LIN {X 26.609, Y 67.769, Z 160.75, A 0, B 90, C 0, E1 0, E2 0, E3 0, E4 0} C_DIS
LIN {X 29.432, Y 66.695, Z 160.75, A 0, B 90, C 0, E1 0, E2 0, E3 0, E4 0} C_DIS
LIN {X 32.336, Y 65.861, Z 160.75, A 0, B 90, C 0, E1 0, E2 0, E3 0, E4 0} C_DIS
LIN {X 35.293, Y 65.239, Z 160.75, A 0, B 90, C 0, E1 0, E2 0, E3 0, E4 0} C_DIS
LIN {X 38.28, Y 64.777, Z 160.75, A 0, B 90, C 0, E1 0, E2 0, E3 0, E4 0} C_DIS
LIN {X 41.281, Y 64.423, Z 160.75, A 0, B 90, C 0, E1 0, E2 0, E3 0, E4 0} C_DIS
LIN {X 44.288, Y 64.127, Z 160.75, A 0, B 90, C 0, E1 0, E2 0, E3 0, E4 0} C_DIS
LIN {X 47.298, Y 63.846, Z 160.75, A 0, B 90, C 0, E1 0, E2 0, E3 0, E4 0} C_DIS
LIN {X 50.305, Y 63.548, Z 160.75, A 0, B 90, C 0, E1 0, E2 0, E3 0, E4 0} C_DIS
LIN {X 53.308, Y 63.205, Z 160.75, A 0, B 90, C 0, E1 0, E2 0, E3 0, E4 0} C_DIS
LIN {X 56.302, Y 62.795, Z 160.75, A 0, B 90, C 0, E1 0, E2 0, E3 0, E4 0} C_DIS
LIN {X 59.283, Y 62.3, Z 160.75, A 0, B 90, C 0, E1 0, E2 0, E3 0, E4 0} C_DIS
LIN {X 62.245, Y 61.704, Z 160.75, A 0, B 90, C 0, E1 0, E2 0, E3 0, E4 0} C_DIS
LIN {X 65.182, Y 60.99, Z 160.75, A 0, B 90, C 0, E1 0, E2 0, E3 0, E4 0} C_DIS
LIN {X 68.084, Y 60.146, Z 160.75, A 0, B 90, C 0, E1 0, E2 0, E3 0, E4 0} C_DIS
LIN {X 70.939, Y 59.158, Z 160.75, A 0, B 90, C 0, E1 0, E2 0, E3 0, E4 0} C_DIS
LIN {X 73.737, Y 58.015, Z 160.75, A 0, B 90, C 0, E1 0, E2 0, E3 0, E4 0} C_DIS
LIN {X 76.46, Y 56.707, Z 160.75, A 0, B 90, C 0, E1 0, E2 0, E3 0, E4 0} C_DIS
LIN {X 79.094, Y 55.225, Z 160.75, A 0, B 90, C 0, E1 0, E2 0, E3 0, E4 0} C_DIS
LIN {X 81.618, Y 53.564, Z 160.75, A 0, B 90, C 0, E1 0, E2 0, E3 0, E4 0} C_DIS
LIN {X 84.013, Y 51.722, Z 160.75, A 0, B 90, C 0, E1 0, E2 0, E3 0, E4 0} C_DIS
LIN {X 86.258, Y 49.701, Z 160.75, A 0, B 90, C 0, E1 0, E2 0, E3 0, E4 0} C_DIS
LIN {X 88.328, Y 47.5, Z 160.75, A 0, B 90, C 0, E1 0, E2 0, E3 0, E4 0} C_DIS
LIN {X 90.195, Y 45.125, Z 160.75, A 0, B 90, C 0, E1 0, E2 0, E3 0, E4 0} C_DIS
LIN {X 91.836, Y 42.588, Z 160.75, A 0, B 90, C 0, E1 0, E2 0, E3 0, E4 0} C_DIS
LIN {X 93.229, Y 39.908, Z 160.75, A 0, B 90, C 0, E1 0, E2 0, E3 0, E4 0} C_DIS
LIN {X 94.359, Y 37.106, Z 160.75, A 0, B 90, C 0, E1 0, E2 0, E3 0, E4 0} C_DIS
LIN {X 95.213, Y 34.208, Z 160.75, A 0, B 90, C 0, E1 0, E2 0, E3 0, E4 0} C_DIS
LIN {X 95.79, Y 31.243, Z 160.75, A 0, B 90, C 0, E1 0, E2 0, E3 0, E4 0} C_DIS
LIN {X 96.091, Y 28.237, Z 160.75, A 0, B 90, C 0, E1 0, E2 0, E3 0, E4 0} C_DIS
LIN {X 96.125, Y 25.216, Z 160.75, A 0, B 90, C 0, E1 0, E2 0, E3 0, E4 0} C_DIS
LIN {X 95.904, Y 22.202, Z 160.75, A 0, B 90, C 0, E1 0, E2 0, E3 0, E4 0} C_DIS
LIN {X 95.444, Y 19.216, Z 160.75, A 0, B 90, C 0, E1 0, E2 0, E3 0, E4 0} C_DIS
LIN {X 94.762, Y 16.273, Z 160.75, A 0, B 90, C 0, E1 0, E2 0, E3 0, E4 0} C_DIS
LIN {X 93.877, Y 13.384, Z 160.75, A 0, B 90, C 0, E1 0, E2 0, E3 0, E4 0} C_DIS
LIN {X 92.806, Y 10.558, Z 160.75, A 0, B 90, C 0, E1 0, E2 0, E3 0, E4 0} C_DIS
LIN {X 91.571, Y 7.8, Z 160.75, A 0, B 90, C 0, E1 0, E2 0, E3 0, E4 0} C_DIS
LIN {X 90.195, Y 5.11, Z 160.75, A 0, B 90, C 0, E1 0, E2 0, E3 0, E4 0} C_DIS
LIN {X 88.691, Y 2.489, Z 160.75, A 0, B 90, C 0, E1 0, E2 0, E3 0, E4 0} C_DIS
LIN {X 87.109, Y 0, Z 160.75, A 0, B 90, C 0, E1 0, E2 0, E3 0, E4 0} C_DIS
LIN {X 85.255, Y -2.058, Z 160.75, A 0, B 90, C 0, E1 0, E2 0, E3 0, E4 0} C_DIS
LIN {X 83.459, Y -4.487, Z 160.75, A 0, B 90, C 0, E1 0, E2 0, E3 0, E4 0} C_DIS
LIN {X 81.625, Y -6.889, Z 160.75, A 0, B 90, C 0, E1 0, E2 0, E3 0, E4 0} C_DIS
LIN {X 79.745, Y -9.255, Z 160.75, A 0, B 90, C 0, E1 0, E2 0, E3 0, E4 0} C_DIS
LIN {X 77.844, Y -11.605, Z 160.75, A 0, B 90, C 0, E1 0, E2 0, E3 0, E4 0} C_DIS
LIN {X 75.949, Y -13.959, Z 160.75, A 0, B 90, C 0, E1 0, E2 0, E3 0, E4 0} C_DIS
LIN {X 74.087, Y -16.339, Z 160.75, A 0, B 90, C 0, E1 0, E2 0, E3 0, E4 0} C_DIS
LIN {X 72.293, Y -18.771, Z 160.75, A 0, B 90, C 0, E1 0, E2 0, E3 0, E4 0} C_DIS
LIN {X 70.608, Y -21.279, Z 160.75, A 0, B 90, C 0, E1 0, E2 0, E3 0, E4 0} C_DIS
LIN {X 69.084, Y -23.889, Z 160.75, A 0, B 90, C 0, E1 0, E2 0, E3 0, E4 0} C_DIS
LIN {X 67.769, Y -26.609, Z 160.75, A 0, B 90, C 0, E1 0, E2 0, E3 0, E4 0} C_DIS
LIN {X 66.695, Y -29.432, Z 160.75, A 0, B 90, C 0, E1 0, E2 0, E3 0, E4 0} C_DIS
LIN {X 65.861, Y -32.336, Z 160.75, A 0, B 90, C 0, E1 0, E2 0, E3 0, E4 0} C_DIS
LIN {X 65.239, Y -35.293, Z 160.75, A 0, B 90, C 0, E1 0, E2 0, E3 0, E4 0} C_DIS
LIN {X 64.777, Y -38.28, Z 160.75, A 0, B 90, C 0, E1 0, E2 0, E3 0, E4 0} C_DIS
LIN {X 64.423, Y -41.281, Z 160.75, A 0, B 90, C 0, E1 0, E2 0, E3 0, E4 0} C_DIS
LIN {X 64.127, Y -44.288, Z 160.75, A 0, B 90, C 0, E1 0, E2 0, E3 0, E4 0} C_DIS
LIN {X 63.846, Y -47.298, Z 160.75, A 0, B 90, C 0, E1 0, E2 0, E3 0, E4 0} C_DIS
LIN {X 63.548, Y -50.305, Z 160.75, A 0, B 90, C 0, E1 0, E2 0, E3 0, E4 0} C_DIS
LIN {X 63.205, Y -53.308, Z 160.75, A 0, B 90, C 0, E1 0, E2 0, E3 0, E4 0} C_DIS
LIN {X 62.795, Y -56.302, Z 160.75, A 0, B 90, C 0, E1 0, E2 0, E3 0, E4 0} C_DIS
LIN {X 62.3, Y -59.283, Z 160.75, A 0, B 90, C 0, E1 0, E2 0, E3 0, E4 0} C_DIS
LIN {X 61.704, Y -62.245, Z 160.75, A 0, B 90, C 0, E1 0, E2 0, E3 0, E4 0} C_DIS
LIN {X 60.99, Y -65.182, Z 160.75, A 0, B 90, C 0, E1 0, E2 0, E3 0, E4 0} C_DIS
LIN {X 60.146, Y -68.084, Z 160.75, A 0, B 90, C 0, E1 0, E2 0, E3 0, E4 0} C_DIS
LIN {X 59.158, Y -70.939, Z 160.75, A 0, B 90, C 0, E1 0, E2 0, E3 0, E4 0} C_DIS
LIN {X 58.015, Y -73.737, Z 160.75, A 0, B 90, C 0, E1 0, E2 0, E3 0, E4 0} C_DIS
LIN {X 56.707, Y -76.46, Z 160.75, A 0, B 90, C 0, E1 0, E2 0, E3 0, E4 0} C_DIS
LIN {X 55.225, Y -79.094, Z 160.75, A 0, B 90, C 0, E1 0, E2 0, E3 0, E4 0} C_DIS
LIN {X 53.564, Y -81.618, Z 160.75, A 0, B 90, C 0, E1 0, E2 0, E3 0, E4 0} C_DIS
LIN {X 51.722, Y -84.013, Z 160.75, A 0, B 90, C 0, E1 0, E2 0, E3 0, E4 0} C_DIS
LIN {X 49.701, Y -86.258, Z 160.75, A 0, B 90, C 0, E1 0, E2 0, E3 0, E4 0} C_DIS
LIN {X 47.5, Y -88.328, Z 160.75, A 0, B 90, C 0, E1 0, E2 0, E3 0, E4 0} C_DIS
LIN {X 45.125, Y -90.195, Z 160.75, A 0, B 90, C 0, E1 0, E2 0, E3 0, E4 0} C_DIS
LIN {X 42.588, Y -91.836, Z 160.75, A 0, B 90, C 0, E1 0, E2 0, E3 0, E4 0} C_DIS
LIN {X 39.908, Y -93.229, Z 160.75, A 0, B 90, C 0, E1 0, E2 0, E3 0, E4 0} C_DIS
LIN {X 37.106, Y -94.359, Z 160.75, A 0, B 90, C 0, E1 0, E2 0, E3 0, E4 0} C_DIS
LIN {X 34.208, Y -95.213, Z 160.75, A 0, B 90, C 0, E1 0, E2 0, E3 0, E4 0} C_DIS
LIN {X 31.243, Y -95.79, Z 160.75, A 0, B 90, C 0, E1 0, E2 0, E3 0, E4 0} C_DIS
LIN {X 28.237, Y -96.091, Z 160.75, A 0, B 90, C 0, E1 0, E2 0, E3 0, E4 0} C_DIS
LIN {X 25.216, Y -96.125, Z 160.75, A 0, B 90, C 0, E1 0, E2 0, E3 0, E4 0} C_DIS
LIN {X 22.202, Y -95.904, Z 160.75, A 0, B 90, C 0, E1 0, E2 0, E3 0, E4 0} C_DIS
LIN {X 19.216, Y -95.444, Z 160.75, A 0, B 90, C 0, E1 0, E2 0, E3 0, E4 0} C_DIS
LIN {X 16.273, Y -94.762, Z 160.75, A 0, B 90, C 0, E1 0, E2 0, E3 0, E4 0} C_DIS
LIN {X 13.384, Y -93.877, Z 160.75, A 0, B 90, C 0, E1 0, E2 0, E3 0, E4 0} C_DIS
LIN {X 10.558, Y -92.806, Z 160.75, A 0, B 90, C 0, E1 0, E2 0, E3 0, E4 0} C_DIS
LIN {X 7.8, Y -91.571, Z 160.75, A 0, B 90, C 0, E1 0, E2 0, E3 0, E4 0} C_DIS
LIN {X 5.11, Y -90.195, Z 160.75, A 0, B 90, C 0, E1 0, E2 0, E3 0, E4 0} C_DIS
LIN {X 2.489, Y -88.691, Z 160.75, A 0, B 90, C 0, E1 0, E2 0, E3 0, E4 0} C_DIS
LIN {X 0, Y -87.109, Z 160.75, A 0, B 90, C 0, E1 0, E2 0, E3 0, E4 0} C_DIS
LIN {X -2.058, Y -85.255, Z 160.75, A 0, B 90, C 0, E1 0, E2 0, E3 0, E4 0} C_DIS
LIN {X -4.487, Y -83.459, Z 160.75, A 0, B 90, C 0, E1 0, E2 0, E3 0, E4 0} C_DIS
LIN {X -6.889, Y -81.625, Z 160.75, A 0, B 90, C 0, E1 0, E2 0, E3 0, E4 0} C_DIS
LIN {X -9.255, Y -79.745, Z 160.75, A 0, B 90, C 0, E1 0, E2 0, E3 0, E4 0} C_DIS
LIN {X -11.605, Y -77.844, Z 160.75, A 0, B 90, C 0, E1 0, E2 0, E3 0, E4 0} C_DIS
LIN {X -13.959, Y -75.949, Z 160.75, A 0, B 90, C 0, E1 0, E2 0, E3 0, E4 0} C_DIS
LIN {X -16.339, Y -74.087, Z 160.75, A 0, B 90, C 0, E1 0, E2 0, E3 0, E4 0} C_DIS
LIN {X -18.771, Y -72.293, Z 160.75, A 0, B 90, C 0, E1 0, E2 0, E3 0, E4 0} C_DIS
LIN {X -21.279, Y -70.608, Z 160.75, A 0, B 90, C 0, E1 0, E2 0, E3 0, E4 0} C_DIS
LIN {X -23.889, Y -69.084, Z 160.75, A 0, B 90, C 0, E1 0, E2 0, E3 0, E4 0} C_DIS
LIN {X -26.609, Y -67.769, Z 160.75, A 0, B 90, C 0, E1 0, E2 0, E3 0, E4 0} C_DIS
LIN {X -29.432, Y -66.695, Z 160.75, A 0, B 90, C 0, E1 0, E2 0, E3 0, E4 0} C_DIS
LIN {X -32.336, Y -65.861, Z 160.75, A 0, B 90, C 0, E1 0, E2 0, E3 0, E4 0} C_DIS
LIN {X -35.293, Y -65.239, Z 160.75, A 0, B 90, C 0, E1 0, E2 0, E3 0, E4 0} C_DIS
LIN {X -38.28, Y -64.777, Z 160.75, A 0, B 90, C 0, E1 0, E2 0, E3 0, E4 0} C_DIS
LIN {X -41.281, Y -64.423, Z 160.75, A 0, B 90, C 0, E1 0, E2 0, E3 0, E4 0} C_DIS
LIN {X -44.288, Y -64.127, Z 160.75, A 0, B 90, C 0, E1 0, E2 0, E3 0, E4 0} C_DIS
LIN {X -47.298, Y -63.846, Z 160.75, A 0, B 90, C 0, E1 0, E2 0, E3 0, E4 0} C_DIS
LIN {X -50.305, Y -63.548, Z 160.75, A 0, B 90, C 0, E1 0, E2 0, E3 0, E4 0} C_DIS
LIN {X -53.308, Y -63.205, Z 160.75, A 0, B 90, C 0, E1 0, E2 0, E3 0, E4 0} C_DIS
LIN {X -56.302, Y -62.795, Z 160.75, A 0, B 90, C 0, E1 0, E2 0, E3 0, E4 0} C_DIS
LIN {X -59.283, Y -62.3, Z 160.75, A 0, B 90, C 0, E1 0, E2 0, E3 0, E4 0} C_DIS
LIN {X -62.245, Y -61.704, Z 160.75, A 0, B 90, C 0, E1 0, E2 0, E3 0, E4 0} C_DIS
LIN {X -65.182, Y -60.99, Z 160.75, A 0, B 90, C 0, E1 0, E2 0, E3 0, E4 0} C_DIS
LIN {X -68.084, Y -60.146, Z 160.75, A 0, B 90, C 0, E1 0, E2 0, E3 0, E4 0} C_DIS
LIN {X -70.939, Y -59.158, Z 160.75, A 0, B 90, C 0, E1 0, E2 0, E3 0, E4 0} C_DIS
LIN {X -73.737, Y -58.015, Z 160.75, A 0, B 90, C 0, E1 0, E2 0, E3 0, E4 0} C_DIS
LIN {X -76.46, Y -56.707, Z 160.75, A 0, B 90, C 0, E1 0, E2 0, E3 0, E4 0} C_DIS
LIN {X -79.094, Y -55.225, Z 160.75, A 0, B 90, C 0, E1 0, E2 0, E3 0, E4 0} C_DIS
LIN {X -81.618, Y -53.564, Z 160.75, A 0, B 90, C 0, E1 0, E2 0, E3 0, E4 0} C_DIS
LIN {X -84.013, Y -51.722, Z 160.75, A 0, B 90, C 0, E1 0, E2 0, E3 0, E4 0} C_DIS
LIN {X -86.258, Y -49.701, Z 160.75, A 0, B 90, C 0, E1 0, E2 0, E3 0, E4 0} C_DIS
LIN {X -88.328, Y -47.5, Z 160.75, A 0, B 90, C 0, E1 0, E2 0, E3 0, E4 0} C_DIS
LIN {X -90.195, Y -45.125, Z 160.75, A 0, B 90, C 0, E1 0, E2 0, E3 0, E4 0} C_DIS
LIN {X -91.836, Y -42.588, Z 160.75, A 0, B 90, C 0, E1 0, E2 0, E3 0, E4 0} C_DIS
LIN {X -93.229, Y -39.908, Z 160.75, A 0, B 90, C 0, E1 0, E2 0, E3 0, E4 0} C_DIS
LIN {X -94.359, Y -37.106, Z 160.75, A 0, B 90, C 0, E1 0, E2 0, E3 0, E4 0} C_DIS
LIN {X -95.213, Y -34.208, Z 160.75, A 0, B 90, C 0, E1 0, E2 0, E3 0, E4 0} C_DIS
LIN {X -95.79, Y -31.243, Z 160.75, A 0, B 90, C 0, E1 0, E2 0, E3 0, E4 0} C_DIS
LIN {X -96.091, Y -28.237, Z 160.75, A 0, B 90, C 0, E1 0, E2 0, E3 0, E4 0} C_DIS
LIN {X -96.125, Y -25.216, Z 160.75, A 0, B 90, C 0, E1 0, E2 0, E3 0, E4 0} C_DIS
LIN {X -95.904, Y -22.202, Z 160.75, A 0, B 90, C 0, E1 0, E2 0, E3 0, E4 0} C_DIS
LIN {X -95.444, Y -19.216, Z 160.75, A 0, B 90, C 0, E1 0, E2 0, E3 0, E4 0} C_DIS
LIN {X -94.762, Y -16.273, Z 160.75, A 0, B 90, C 0, E1 0, E2 0, E3 0, E4 0} C_DIS
LIN {X -93.877, Y -13.384, Z 160.75, A 0, B 90, C 0, E1 0, E2 0, E3 0, E4 0} C_DIS
LIN {X -92.806, Y -10.558, Z 160.75, A 0, B 90, C 0, E1 0, E2 0, E3 0, E4 0} C_DIS
LIN {X -91.571, Y -7.8, Z 160.75, A 0, B 90, C 0, E1 0, E2 0, E3 0, E4 0} C_DIS
LIN {X -90.195, Y -5.11, Z 160.75, A 0, B 90, C 0, E1 0, E2 0, E3 0, E4 0} C_DIS
LIN {X -88.691, Y -2.489, Z 160.75, A 0, B 90, C 0, E1 0, E2 0, E3 0, E4 0} C_DIS
LIN {X -87.509, Y 0, Z 163.25, A 0, B 90, C 0, E1 0, E2 0, E3 0, E4 0} C_DIS
LIN {X -85.636, Y 2.054, Z 163.25, A 0, B 90, C 0, E1 0, E2 0, E3 0, E4 0} C_DIS
LIN {X -83.819, Y 4.483, Z 163.25, A 0, B 90, C 0, E1 0, E2 0, E3 0, E4 0} C_DIS
LIN {X -81.966, Y 6.885, Z 163.25, A 0, B 90, C 0, E1 0, E2 0, E3 0, E4 0} C_DIS
LIN {X -80.069, Y 9.253, Z 163.25, A 0, B 90, C 0, E1 0, E2 0, E3 0, E4 0} C_DIS
LIN {X -78.156, Y 11.608, Z 163.25, A 0, B 90, C 0, E1 0, E2 0, E3 0, E4 0} C_DIS
LIN {X -76.258, Y 13.975, Z 163.25, A 0, B 90, C 0, E1 0, E2 0, E3 0, E4 0} C_DIS
LIN {X -74.403, Y 16.376, Z 163.25, A 0, B 90, C 0, E1 0, E2 0, E3 0, E4 0} C_DIS
LIN {X -72.622, Y 18.832, Z 163.25, A 0, B 90, C 0, E1 0, E2 0, E3 0, E4 0} C_DIS
LIN {X -70.954, Y 21.366, Z 163.25, A 0, B 90, C 0, E1 0, E2 0, E3 0, E4 0} C_DIS
LIN {X -69.45, Y 24.001, Z 163.25, A 0, B 90, C 0, E1 0, E2 0, E3 0, E4 0} C_DIS
LIN {X -68.156, Y 26.744, Z 163.25, A 0, B 90, C 0, E1 0, E2 0, E3 0, E4 0} C_DIS
LIN {X -67.106, Y 29.59, Z 163.25, A 0, B 90, C 0, E1 0, E2 0, E3 0, E4 0} C_DIS
LIN {X -66.295, Y 32.513, Z 163.25, A 0, B 90, C 0, E1 0, E2 0, E3 0, E4 0} C_DIS
LIN {X -65.695, Y 35.486, Z 163.25, A 0, B 90, C 0, E1 0, E2 0, E3 0, E4 0} C_DIS
LIN {X -65.252, Y 38.488, Z 163.25, A 0, B 90, C 0, E1 0, E2 0, E3 0, E4 0} C_DIS
LIN {X -64.912, Y 41.503, Z 163.25, A 0, B 90, C 0, E1 0, E2 0, E3 0, E4 0} C_DIS
LIN {X -64.622, Y 44.523, Z 163.25, A 0, B 90, C 0, E1 0, E2 0, E3 0, E4 0} C_DIS
LIN {X -64.34, Y 47.544, Z 163.25, A 0, B 90, C 0, E1 0, E2 0, E3 0, E4 0} C_DIS
LIN {X -64.029, Y 50.562, Z 163.25, A 0, B 90, C 0, E1 0, E2 0, E3 0, E4 0} C_DIS
LIN {X -63.665, Y 53.574, Z 163.25, A 0, B 90, C 0, E1 0, E2 0, E3 0, E4 0} C_DIS
LIN {X -63.229, Y 56.577, Z 163.25, A 0, B 90, C 0, E1 0, E2 0, E3 0, E4 0} C_DIS
LIN {X -62.704, Y 59.565, Z 163.25, A 0, B 90, C 0, E1 0, E2 0, E3 0, E4 0} C_DIS
LIN {X -62.074, Y 62.533, Z 163.25, A 0, B 90, C 0, E1 0, E2 0, E3 0, E4 0} C_DIS
LIN {X -61.326, Y 65.473, Z 163.25, A 0, B 90, C 0, E1 0, E2 0, E3 0, E4 0} C_DIS
LIN {X -60.446, Y 68.376, Z 163.25, A 0, B 90, C 0, E1 0, E2 0, E3 0, E4 0} C_DIS
LIN {X -59.421, Y 71.232, Z 163.25, A 0, B 90, C 0, E1 0, E2 0, E3 0, E4 0} C_DIS
LIN {X -58.24, Y 74.026, Z 163.25, A 0, B 90, C 0, E1 0, E2 0, E3 0, E4 0} C_DIS
LIN {X -56.893, Y 76.744, Z 163.25, A 0, B 90, C 0, E1 0, E2 0, E3 0, E4 0} C_DIS
LIN {X -55.374, Y 79.37, Z 163.25, A 0, B 90, C 0, E1 0, E2 0, E3 0, E4 0} C_DIS
LIN {X -53.681, Y 81.887, Z 163.25, A 0, B 90, C 0, E1 0, E2 0, E3 0, E4 0} C_DIS
LIN {X -51.817, Y 84.28, Z 163.25, A 0, B 90, C 0, E1 0, E2 0, E3 0, E4 0} C_DIS
LIN {X -49.786, Y 86.534, Z 163.25, A 0, B 90, C 0, E1 0, E2 0, E3 0, E4 0} C_DIS
LIN {X -47.585, Y 88.62, Z 163.25, A 0, B 90, C 0, E1 0, E2 0, E3 0, E4 0} C_DIS
LIN {X -45.213, Y 90.511, Z 163.25, A 0, B 90, C 0, E1 0, E2 0, E3 0, E4 0} C_DIS
LIN {X -42.679, Y 92.178, Z 163.25, A 0, B 90, C 0, E1 0, E2 0, E3 0, E4 0} C_DIS
LIN {X -40, Y 93.599, Z 163.25, A 0, B 90, C 0, E1 0, E2 0, E3 0, E4 0} C_DIS
LIN {X -37.197, Y 94.757, Z 163.25, A 0, B 90, C 0, E1 0, E2 0, E3 0, E4 0} C_DIS
LIN {X -34.295, Y 95.639, Z 163.25, A 0, B 90, C 0, E1 0, E2 0, E3 0, E4 0} C_DIS
LIN {X -31.322, Y 96.242, Z 163.25, A 0, B 90, C 0, E1 0, E2 0, E3 0, E4 0} C_DIS
LIN {X -28.307, Y 96.566, Z 163.25, A 0, B 90, C 0, E1 0, E2 0, E3 0, E4 0} C_DIS
LIN {X -25.274, Y 96.62, Z 163.25, A 0, B 90, C 0, E1 0, E2 0, E3 0, E4 0} C_DIS
LIN {X -22.248, Y 96.413, Z 163.25, A 0, B 90, C 0, E1 0, E2 0, E3 0, E4 0} C_DIS
LIN {X -19.248, Y 95.96, Z 163.25, A 0, B 90, C 0, E1 0, E2 0, E3 0, E4 0} C_DIS
LIN {X -16.293, Y 95.276, Z 163.25, A 0, B 90, C 0, E1 0, E2 0, E3 0, E4 0} C_DIS
LIN {X -13.395, Y 94.381, Z 163.25, A 0, B 90, C 0, E1 0, E2 0, E3 0, E4 0} C_DIS
LIN {X -10.563, Y 93.294, Z 163.25, A 0, B 90, C 0, E1 0, E2 0, E3 0, E4 0} C_DIS
LIN {X -7.801, Y 92.039, Z 163.25, A 0, B 90, C 0, E1 0, E2 0, E3 0, E4 0} C_DIS
LIN {X -5.108, Y 90.641, Z 163.25, A 0, B 90, C 0, E1 0, E2 0, E3 0, E4 0} C_DIS
LIN {X -2.488, Y 89.113, Z 163.25, A 0, B 90, C 0, E1 0, E2 0, E3 0, E4 0} C_DIS
LIN {X 0, Y 87.509, Z 163.25, A 0, B 90, C 0, E1 0, E2 0, E3 0, E4 0} C_DIS
LIN {X 2.054, Y 85.636, Z 163.25, A 0, B 90, C 0, E1 0, E2 0, E3 0, E4 0} C_DIS
LIN {X 4.483, Y 83.819, Z 163.25, A 0, B 90, C 0, E1 0, E2 0, E3 0, E4 0} C_DIS
LIN {X 6.885, Y 81.966, Z 163.25, A 0, B 90, C 0, E1 0, E2 0, E3 0, E4 0} C_DIS
LIN {X 9.253, Y 80.069, Z 163.25, A 0, B 90, C 0, E1 0, E2 0, E3 0, E4 0} C_DIS
LIN {X 11.608, Y 78.156, Z 163.25, A 0, B 90, C 0, E1 0, E2 0, E3 0, E4 0} C_DIS
LIN {X 13.975, Y 76.258, Z 163.25, A 0, B 90, C 0, E1 0, E2 0, E3 0, E4 0} C_DIS
LIN {X 16.376, Y 74.403, Z 163.25, A 0, B 90, C 0, E1 0, E2 0, E3 0, E4 0} C_DIS
LIN {X 18.832, Y 72.622, Z 163.25, A 0, B 90, C 0, E1 0, E2 0, E3 0, E4 0} C_DIS
LIN {X 21.366, Y 70.954, Z 163.25, A 0, B 90, C 0, E1 0, E2 0, E3 0, E4 0} C_DIS
LIN {X 24.001, Y 69.45, Z 163.25, A 0, B 90, C 0, E1 0, E2 0, E3 0, E4 0} C_DIS
LIN {X 26.744, Y 68.156, Z 163.25, A 0, B 90, C 0, E1 0, E2 0, E3 0, E4 0} C_DIS
LIN {X 29.59, Y 67.106, Z 163.25, A 0, B 90, C 0, E1 0, E2 0, E3 0, E4 0} C_DIS
LIN {X 32.513, Y 66.295, Z 163.25, A 0, B 90, C 0, E1 0, E2 0, E3 0, E4 0} C_DIS
LIN {X 35.486, Y 65.695, Z 163.25, A 0, B 90, C 0, E1 0, E2 0, E3 0, E4 0} C_DIS
LIN {X 38.488, Y 65.252, Z 163.25, A 0, B 90, C 0, E1 0, E2 0, E3 0, E4 0} C_DIS
LIN {X 41.503, Y 64.912, Z 163.25, A 0, B 90, C 0, E1 0, E2 0, E3 0, E4 0} C_DIS
LIN {X 44.523, Y 64.622, Z 163.25, A 0, B 90, C 0, E1 0, E2 0, E3 0, E4 0} C_DIS
LIN {X 47.544, Y 64.34, Z 163.25, A 0, B 90, C 0, E1 0, E2 0, E3 0, E4 0} C_DIS
LIN {X 50.562, Y 64.029, Z 163.25, A 0, B 90, C 0, E1 0, E2 0, E3 0, E4 0} C_DIS
LIN {X 53.574, Y 63.665, Z 163.25, A 0, B 90, C 0, E1 0, E2 0, E3 0, E4 0} C_DIS
LIN {X 56.577, Y 63.229, Z 163.25, A 0, B 90, C 0, E1 0, E2 0, E3 0, E4 0} C_DIS
LIN {X 59.565, Y 62.704, Z 163.25, A 0, B 90, C 0, E1 0, E2 0, E3 0, E4 0} C_DIS
LIN {X 62.533, Y 62.074, Z 163.25, A 0, B 90, C 0, E1 0, E2 0, E3 0, E4 0} C_DIS
LIN {X 65.473, Y 61.326, Z 163.25, A 0, B 90, C 0, E1 0, E2 0, E3 0, E4 0} C_DIS
LIN {X 68.376, Y 60.446, Z 163.25, A 0, B 90, C 0, E1 0, E2 0, E3 0, E4 0} C_DIS
LIN {X 71.232, Y 59.421, Z 163.25, A 0, B 90, C 0, E1 0, E2 0, E3 0, E4 0} C_DIS
LIN {X 74.026, Y 58.24, Z 163.25, A 0, B 90, C 0, E1 0, E2 0, E3 0, E4 0} C_DIS
LIN {X 76.744, Y 56.893, Z 163.25, A 0, B 90, C 0, E1 0, E2 0, E3 0, E4 0} C_DIS
LIN {X 79.37, Y 55.374, Z 163.25, A 0, B 90, C 0, E1 0, E2 0, E3 0, E4 0} C_DIS
LIN {X 81.887, Y 53.681, Z 163.25, A 0, B 90, C 0, E1 0, E2 0, E3 0, E4 0} C_DIS
LIN {X 84.28, Y 51.817, Z 163.25, A 0, B 90, C 0, E1 0, E2 0, E3 0, E4 0} C_DIS
LIN {X 86.534, Y 49.786, Z 163.25, A 0, B 90, C 0, E1 0, E2 0, E3 0, E4 0} C_DIS
LIN {X 88.62, Y 47.585, Z 163.25, A 0, B 90, C 0, E1 0, E2 0, E3 0, E4 0} C_DIS
LIN {X 90.511, Y 45.213, Z 163.25, A 0, B 90, C 0, E1 0, E2 0, E3 0, E4 0} C_DIS
LIN {X 92.178, Y 42.679, Z 163.25, A 0, B 90, C 0, E1 0, E2 0, E3 0, E4 0} C_DIS
LIN {X 93.599, Y 40, Z 163.25, A 0, B 90, C 0, E1 0, E2 0, E3 0, E4 0} C_DIS
LIN {X 94.757, Y 37.197, Z 163.25, A 0, B 90, C 0, E1 0, E2 0, E3 0, E4 0} C_DIS
LIN {X 95.639, Y 34.295, Z 163.25, A 0, B 90, C 0, E1 0, E2 0, E3 0, E4 0} C_DIS
LIN {X 96.242, Y 31.322, Z 163.25, A 0, B 90, C 0, E1 0, E2 0, E3 0, E4 0} C_DIS
LIN {X 96.566, Y 28.307, Z 163.25, A 0, B 90, C 0, E1 0, E2 0, E3 0, E4 0} C_DIS
LIN {X 96.62, Y 25.274, Z 163.25, A 0, B 90, C 0, E1 0, E2 0, E3 0, E4 0} C_DIS
LIN {X 96.413, Y 22.248, Z 163.25, A 0, B 90, C 0, E1 0, E2 0, E3 0, E4 0} C_DIS
LIN {X 95.96, Y 19.248, Z 163.25, A 0, B 90, C 0, E1 0, E2 0, E3 0, E4 0} C_DIS
LIN {X 95.276, Y 16.293, Z 163.25, A 0, B 90, C 0, E1 0, E2 0, E3 0, E4 0} C_DIS
LIN {X 94.381, Y 13.395, Z 163.25, A 0, B 90, C 0, E1 0, E2 0, E3 0, E4 0} C_DIS
LIN {X 93.294, Y 10.563, Z 163.25, A 0, B 90, C 0, E1 0, E2 0, E3 0, E4 0} C_DIS
LIN {X 92.039, Y 7.801, Z 163.25, A 0, B 90, C 0, E1 0, E2 0, E3 0, E4 0} C_DIS
LIN {X 90.641, Y 5.108, Z 163.25, A 0, B 90, C 0, E1 0, E2 0, E3 0, E4 0} C_DIS
LIN {X 89.113, Y 2.488, Z 163.25, A 0, B 90, C 0, E1 0, E2 0, E3 0, E4 0} C_DIS
LIN {X 87.509, Y 0, Z 163.25, A 0, B 90, C 0, E1 0, E2 0, E3 0, E4 0} C_DIS
LIN {X 85.636, Y -2.054, Z 163.25, A 0, B 90, C 0, E1 0, E2 0, E3 0, E4 0} C_DIS
LIN {X 83.819, Y -4.483, Z 163.25, A 0, B 90, C 0, E1 0, E2 0, E3 0, E4 0} C_DIS
LIN {X 81.966, Y -6.885, Z 163.25, A 0, B 90, C 0, E1 0, E2 0, E3 0, E4 0} C_DIS
LIN {X 80.069, Y -9.253, Z 163.25, A 0, B 90, C 0, E1 0, E2 0, E3 0, E4 0} C_DIS
LIN {X 78.156, Y -11.608, Z 163.25, A 0, B 90, C 0, E1 0, E2 0, E3 0, E4 0} C_DIS
LIN {X 76.258, Y -13.975, Z 163.25, A 0, B 90, C 0, E1 0, E2 0, E3 0, E4 0} C_DIS
LIN {X 74.403, Y -16.376, Z 163.25, A 0, B 90, C 0, E1 0, E2 0, E3 0, E4 0} C_DIS
LIN {X 72.622, Y -18.832, Z 163.25, A 0, B 90, C 0, E1 0, E2 0, E3 0, E4 0} C_DIS
LIN {X 70.954, Y -21.366, Z 163.25, A 0, B 90, C 0, E1 0, E2 0, E3 0, E4 0} C_DIS
LIN {X 69.45, Y -24.001, Z 163.25, A 0, B 90, C 0, E1 0, E2 0, E3 0, E4 0} C_DIS
LIN {X 68.156, Y -26.744, Z 163.25, A 0, B 90, C 0, E1 0, E2 0, E3 0, E4 0} C_DIS
LIN {X 67.106, Y -29.59, Z 163.25, A 0, B 90, C 0, E1 0, E2 0, E3 0, E4 0} C_DIS
LIN {X 66.295, Y -32.513, Z 163.25, A 0, B 90, C 0, E1 0, E2 0, E3 0, E4 0} C_DIS
LIN {X 65.695, Y -35.486, Z 163.25, A 0, B 90, C 0, E1 0, E2 0, E3 0, E4 0} C_DIS
LIN {X 65.252, Y -38.488, Z 163.25, A 0, B 90, C 0, E1 0, E2 0, E3 0, E4 0} C_DIS
LIN {X 64.912, Y -41.503, Z 163.25, A 0, B 90, C 0, E1 0, E2 0, E3 0, E4 0} C_DIS
LIN {X 64.622, Y -44.523, Z 163.25, A 0, B 90, C 0, E1 0, E2 0, E3 0, E4 0} C_DIS
LIN {X 64.34, Y -47.544, Z 163.25, A 0, B 90, C 0, E1 0, E2 0, E3 0, E4 0} C_DIS
LIN {X 64.029, Y -50.562, Z 163.25, A 0, B 90, C 0, E1 0, E2 0, E3 0, E4 0} C_DIS
LIN {X 63.665, Y -53.574, Z 163.25, A 0, B 90, C 0, E1 0, E2 0, E3 0, E4 0} C_DIS
LIN {X 63.229, Y -56.577, Z 163.25, A 0, B 90, C 0, E1 0, E2 0, E3 0, E4 0} C_DIS
LIN {X 62.704, Y -59.565, Z 163.25, A 0, B 90, C 0, E1 0, E2 0, E3 0, E4 0} C_DIS
LIN {X 62.074, Y -62.533, Z 163.25, A 0, B 90, C 0, E1 0, E2 0, E3 0, E4 0} C_DIS
LIN {X 61.326, Y -65.473, Z 163.25, A 0, B 90, C 0, E1 0, E2 0, E3 0, E4 0} C_DIS
LIN {X 60.446, Y -68.376, Z 163.25, A 0, B 90, C 0, E1 0, E2 0, E3 0, E4 0} C_DIS
LIN {X 59.421, Y -71.232, Z 163.25, A 0, B 90, C 0, E1 0, E2 0, E3 0, E4 0} C_DIS
LIN {X 58.24, Y -74.026, Z 163.25, A 0, B 90, C 0, E1 0, E2 0, E3 0, E4 0} C_DIS
LIN {X 56.893, Y -76.744, Z 163.25, A 0, B 90, C 0, E1 0, E2 0, E3 0, E4 0} C_DIS
LIN {X 55.374, Y -79.37, Z 163.25, A 0, B 90, C 0, E1 0, E2 0, E3 0, E4 0} C_DIS
LIN {X 53.681, Y -81.887, Z 163.25, A 0, B 90, C 0, E1 0, E2 0, E3 0, E4 0} C_DIS
LIN {X 51.817, Y -84.28, Z 163.25, A 0, B 90, C 0, E1 0, E2 0, E3 0, E4 0} C_DIS
LIN {X 49.786, Y -86.534, Z 163.25, A 0, B 90, C 0, E1 0, E2 0, E3 0, E4 0} C_DIS
LIN {X 47.585, Y -88.62, Z 163.25, A 0, B 90, C 0, E1 0, E2 0, E3 0, E4 0} C_DIS
LIN {X 45.213, Y -90.511, Z 163.25, A 0, B 90, C 0, E1 0, E2 0, E3 0, E4 0} C_DIS
LIN {X 42.679, Y -92.178, Z 163.25, A 0, B 90, C 0, E1 0, E2 0, E3 0, E4 0} C_DIS
LIN {X 40, Y -93.599, Z 163.25, A 0, B 90, C 0, E1 0, E2 0, E3 0, E4 0} C_DIS
LIN {X 37.197, Y -94.757, Z 163.25, A 0, B 90, C 0, E1 0, E2 0, E3 0, E4 0} C_DIS
LIN {X 34.295, Y -95.639, Z 163.25, A 0, B 90, C 0, E1 0, E2 0, E3 0, E4 0} C_DIS
LIN {X 31.322, Y -96.242, Z 163.25, A 0, B 90, C 0, E1 0, E2 0, E3 0, E4 0} C_DIS
LIN {X 28.307, Y -96.566, Z 163.25, A 0, B 90, C 0, E1 0, E2 0, E3 0, E4 0} C_DIS
LIN {X 25.274, Y -96.62, Z 163.25, A 0, B 90, C 0, E1 0, E2 0, E3 0, E4 0} C_DIS
LIN {X 22.248, Y -96.413, Z 163.25, A 0, B 90, C 0, E1 0, E2 0, E3 0, E4 0} C_DIS
LIN {X 19.248, Y -95.96, Z 163.25, A 0, B 90, C 0, E1 0, E2 0, E3 0, E4 0} C_DIS
LIN {X 16.293, Y -95.276, Z 163.25, A 0, B 90, C 0, E1 0, E2 0, E3 0, E4 0} C_DIS
LIN {X 13.395, Y -94.381, Z 163.25, A 0, B 90, C 0, E1 0, E2 0, E3 0, E4 0} C_DIS
LIN {X 10.563, Y -93.294, Z 163.25, A 0, B 90, C 0, E1 0, E2 0, E3 0, E4 0} C_DIS
LIN {X 7.801, Y -92.039, Z 163.25, A 0, B 90, C 0, E1 0, E2 0, E3 0, E4 0} C_DIS
LIN {X 5.108, Y -90.641, Z 163.25, A 0, B 90, C 0, E1 0, E2 0, E3 0, E4 0} C_DIS
LIN {X 2.488, Y -89.113, Z 163.25, A 0, B 90, C 0, E1 0, E2 0, E3 0, E4 0} C_DIS
LIN {X 0, Y -87.509, Z 163.25, A 0, B 90, C 0, E1 0, E2 0, E3 0, E4 0} C_DIS
LIN {X -2.054, Y -85.636, Z 163.25, A 0, B 90, C 0, E1 0, E2 0, E3 0, E4 0} C_DIS
LIN {X -4.483, Y -83.819, Z 163.25, A 0, B 90, C 0, E1 0, E2 0, E3 0, E4 0} C_DIS
LIN {X -6.885, Y -81.966, Z 163.25, A 0, B 90, C 0, E1 0, E2 0, E3 0, E4 0} C_DIS
LIN {X -9.253, Y -80.069, Z 163.25, A 0, B 90, C 0, E1 0, E2 0, E3 0, E4 0} C_DIS
LIN {X -11.608, Y -78.156, Z 163.25, A 0, B 90, C 0, E1 0, E2 0, E3 0, E4 0} C_DIS
LIN {X -13.975, Y -76.258, Z 163.25, A 0, B 90, C 0, E1 0, E2 0, E3 0, E4 0} C_DIS
LIN {X -16.376, Y -74.403, Z 163.25, A 0, B 90, C 0, E1 0, E2 0, E3 0, E4 0} C_DIS
LIN {X -18.832, Y -72.622, Z 163.25, A 0, B 90, C 0, E1 0, E2 0, E3 0, E4 0} C_DIS
LIN {X -21.366, Y -70.954, Z 163.25, A 0, B 90, C 0, E1 0, E2 0, E3 0, E4 0} C_DIS
LIN {X -24.001, Y -69.45, Z 163.25, A 0, B 90, C 0, E1 0, E2 0, E3 0, E4 0} C_DIS
LIN {X -26.744, Y -68.156, Z 163.25, A 0, B 90, C 0, E1 0, E2 0, E3 0, E4 0} C_DIS
LIN {X -29.59, Y -67.106, Z 163.25, A 0, B 90, C 0, E1 0, E2 0, E3 0, E4 0} C_DIS
LIN {X -32.513, Y -66.295, Z 163.25, A 0, B 90, C 0, E1 0, E2 0, E3 0, E4 0} C_DIS
LIN {X -35.486, Y -65.695, Z 163.25, A 0, B 90, C 0, E1 0, E2 0, E3 0, E4 0} C_DIS
LIN {X -38.488, Y -65.252, Z 163.25, A 0, B 90, C 0, E1 0, E2 0, E3 0, E4 0} C_DIS
LIN {X -41.503, Y -64.912, Z 163.25, A 0, B 90, C 0, E1 0, E2 0, E3 0, E4 0} C_DIS
LIN {X -44.523, Y -64.622, Z 163.25, A 0, B 90, C 0, E1 0, E2 0, E3 0, E4 0} C_DIS
LIN {X -47.544, Y -64.34, Z 163.25, A 0, B 90, C 0, E1 0, E2 0, E3 0, E4 0} C_DIS
LIN {X -50.562, Y -64.029, Z 163.25, A 0, B 90, C 0, E1 0, E2 0, E3 0, E4 0} C_DIS
LIN {X -53.574, Y -63.665, Z 163.25, A 0, B 90, C 0, E1 0, E2 0, E3 0, E4 0} C_DIS
LIN {X -56.577, Y -63.229, Z 163.25, A 0, B 90, C 0, E1 0, E2 0, E3 0, E4 0} C_DIS
LIN {X -59.565, Y -62.704, Z 163.25, A 0, B 90, C 0, E1 0, E2 0, E3 0, E4 0} C_DIS
LIN {X -62.533, Y -62.074, Z 163.25, A 0, B 90, C 0, E1 0, E2 0, E3 0, E4 0} C_DIS
LIN {X -65.473, Y -61.326, Z 163.25, A 0, B 90, C 0, E1 0, E2 0, E3 0, E4 0} C_DIS
LIN {X -68.376, Y -60.446, Z 163.25, A 0, B 90, C 0, E1 0, E2 0, E3 0, E4 0} C_DIS
LIN {X -71.232, Y -59.421, Z 163.25, A 0, B 90, C 0, E1 0, E2 0, E3 0, E4 0} C_DIS
LIN {X -74.026, Y -58.24, Z 163.25, A 0, B 90, C 0, E1 0, E2 0, E3 0, E4 0} C_DIS
LIN {X -76.744, Y -56.893, Z 163.25, A 0, B 90, C 0, E1 0, E2 0, E3 0, E4 0} C_DIS
LIN {X -79.37, Y -55.374, Z 163.25, A 0, B 90, C 0, E1 0, E2 0, E3 0, E4 0} C_DIS
LIN {X -81.887, Y -53.681, Z 163.25, A 0, B 90, C 0, E1 0, E2 0, E3 0, E4 0} C_DIS
LIN {X -84.28, Y -51.817, Z 163.25, A 0, B 90, C 0, E1 0, E2 0, E3 0, E4 0} C_DIS
LIN {X -86.534, Y -49.786, Z 163.25, A 0, B 90, C 0, E1 0, E2 0, E3 0, E4 0} C_DIS
LIN {X -88.62, Y -47.585, Z 163.25, A 0, B 90, C 0, E1 0, E2 0, E3 0, E4 0} C_DIS
LIN {X -90.511, Y -45.213, Z 163.25, A 0, B 90, C 0, E1 0, E2 0, E3 0, E4 0} C_DIS
LIN {X -92.178, Y -42.679, Z 163.25, A 0, B 90, C 0, E1 0, E2 0, E3 0, E4 0} C_DIS
LIN {X -93.599, Y -40, Z 163.25, A 0, B 90, C 0, E1 0, E2 0, E3 0, E4 0} C_DIS
LIN {X -94.757, Y -37.197, Z 163.25, A 0, B 90, C 0, E1 0, E2 0, E3 0, E4 0} C_DIS
LIN {X -95.639, Y -34.295, Z 163.25, A 0, B 90, C 0, E1 0, E2 0, E3 0, E4 0} C_DIS
LIN {X -96.242, Y -31.322, Z 163.25, A 0, B 90, C 0, E1 0, E2 0, E3 0, E4 0} C_DIS
LIN {X -96.566, Y -28.307, Z 163.25, A 0, B 90, C 0, E1 0, E2 0, E3 0, E4 0} C_DIS
LIN {X -96.62, Y -25.274, Z 163.25, A 0, B 90, C 0, E1 0, E2 0, E3 0, E4 0} C_DIS
LIN {X -96.413, Y -22.248, Z 163.25, A 0, B 90, C 0, E1 0, E2 0, E3 0, E4 0} C_DIS
LIN {X -95.96, Y -19.248, Z 163.25, A 0, B 90, C 0, E1 0, E2 0, E3 0, E4 0} C_DIS
LIN {X -95.276, Y -16.293, Z 163.25, A 0, B 90, C 0, E1 0, E2 0, E3 0, E4 0} C_DIS
LIN {X -94.381, Y -13.395, Z 163.25, A 0, B 90, C 0, E1 0, E2 0, E3 0, E4 0} C_DIS
LIN {X -93.294, Y -10.563, Z 163.25, A 0, B 90, C 0, E1 0, E2 0, E3 0, E4 0} C_DIS
LIN {X -92.039, Y -7.801, Z 163.25, A 0, B 90, C 0, E1 0, E2 0, E3 0, E4 0} C_DIS
LIN {X -90.641, Y -5.108, Z 163.25, A 0, B 90, C 0, E1 0, E2 0, E3 0, E4 0} C_DIS
LIN {X -89.113, Y -2.488, Z 163.25, A 0, B 90, C 0, E1 0, E2 0, E3 0, E4 0} C_DIS
LIN {X -87.918, Y 0, Z 165.75, A 0, B 90, C 0, E1 0, E2 0, E3 0, E4 0} C_DIS
LIN {X -86.027, Y 2.051, Z 165.75, A 0, B 90, C 0, E1 0, E2 0, E3 0, E4 0} C_DIS
LIN {X -84.189, Y 4.479, Z 165.75, A 0, B 90, C 0, E1 0, E2 0, E3 0, E4 0} C_DIS
LIN {X -82.316, Y 6.882, Z 165.75, A 0, B 90, C 0, E1 0, E2 0, E3 0, E4 0} C_DIS
LIN {X -80.403, Y 9.252, Z 165.75, A 0, B 90, C 0, E1 0, E2 0, E3 0, E4 0} C_DIS
LIN {X -78.479, Y 11.614, Z 165.75, A 0, B 90, C 0, E1 0, E2 0, E3 0, E4 0} C_DIS
LIN {X -76.578, Y 13.994, Z 165.75, A 0, B 90, C 0, E1 0, E2 0, E3 0, E4 0} C_DIS
LIN {X -74.73, Y 16.416, Z 165.75, A 0, B 90, C 0, E1 0, E2 0, E3 0, E4 0} C_DIS
LIN {X -72.963, Y 18.897, Z 165.75, A 0, B 90, C 0, E1 0, E2 0, E3 0, E4 0} C_DIS
LIN {X -71.314, Y 21.457, Z 165.75, A 0, B 90, C 0, E1 0, E2 0, E3 0, E4 0} C_DIS
LIN {X -69.831, Y 24.118, Z 165.75, A 0, B 90, C 0, E1 0, E2 0, E3 0, E4 0} C_DIS
LIN {X -68.56, Y 26.885, Z 165.75, A 0, B 90, C 0, E1 0, E2 0, E3 0, E4 0} C_DIS
LIN {X -67.534, Y 29.753, Z 165.75, A 0, B 90, C 0, E1 0, E2 0, E3 0, E4 0} C_DIS
LIN {X -66.748, Y 32.695, Z 165.75, A 0, B 90, C 0, E1 0, E2 0, E3 0, E4 0} C_DIS
LIN {X -66.17, Y 35.686, Z 165.75, A 0, B 90, C 0, E1 0, E2 0, E3 0, E4 0} C_DIS
LIN {X -65.747, Y 38.702, Z 165.75, A 0, B 90, C 0, E1 0, E2 0, E3 0, E4 0} C_DIS
LIN {X -65.421, Y 41.731, Z 165.75, A 0, B 90, C 0, E1 0, E2 0, E3 0, E4 0} C_DIS
LIN {X -65.138, Y 44.764, Z 165.75, A 0, B 90, C 0, E1 0, E2 0, E3 0, E4 0} C_DIS
LIN {X -64.853, Y 47.797, Z 165.75, A 0, B 90, C 0, E1 0, E2 0, E3 0, E4 0} C_DIS
LIN {X -64.529, Y 50.826, Z 165.75, A 0, B 90, C 0, E1 0, E2 0, E3 0, E4 0} C_DIS
LIN {X -64.143, Y 53.847, Z 165.75, A 0, B 90, C 0, E1 0, E2 0, E3 0, E4 0} C_DIS
LIN {X -63.679, Y 56.858, Z 165.75, A 0, B 90, C 0, E1 0, E2 0, E3 0, E4 0} C_DIS
LIN {X -63.121, Y 59.853, Z 165.75, A 0, B 90, C 0, E1 0, E2 0, E3 0, E4 0} C_DIS
LIN {X -62.457, Y 62.826, Z 165.75, A 0, B 90, C 0, E1 0, E2 0, E3 0, E4 0} C_DIS
LIN {X -61.673, Y 65.769, Z 165.75, A 0, B 90, C 0, E1 0, E2 0, E3 0, E4 0} C_DIS
LIN {X -60.754, Y 68.673, Z 165.75, A 0, B 90, C 0, E1 0, E2 0, E3 0, E4 0} C_DIS
LIN {X -59.689, Y 71.527, Z 165.75, A 0, B 90, C 0, E1 0, E2 0, E3 0, E4 0} C_DIS
LIN {X -58.468, Y 74.317, Z 165.75, A 0, B 90, C 0, E1 0, E2 0, E3 0, E4 0} C_DIS
LIN {X -57.081, Y 77.029, Z 165.75, A 0, B 90, C 0, E1 0, E2 0, E3 0, E4 0} C_DIS
LIN {X -55.524, Y 79.646, Z 165.75, A 0, B 90, C 0, E1 0, E2 0, E3 0, E4 0} C_DIS
LIN {X -53.797, Y 82.155, Z 165.75, A 0, B 90, C 0, E1 0, E2 0, E3 0, E4 0} C_DIS
LIN {X -51.911, Y 84.547, Z 165.75, A 0, B 90, C 0, E1 0, E2 0, E3 0, E4 0} C_DIS
LIN {X -49.871, Y 86.808, Z 165.75, A 0, B 90, C 0, E1 0, E2 0, E3 0, E4 0} C_DIS
LIN {X -47.669, Y 88.913, Z 165.75, A 0, B 90, C 0, E1 0, E2 0, E3 0, E4 0} C_DIS
LIN {X -45.301, Y 90.827, Z 165.75, A 0, B 90, C 0, E1 0, E2 0, E3 0, E4 0} C_DIS
LIN {X -42.77, Y 92.521, Z 165.75, A 0, B 90, C 0, E1 0, E2 0, E3 0, E4 0} C_DIS
LIN {X -40.093, Y 93.971, Z 165.75, A 0, B 90, C 0, E1 0, E2 0, E3 0, E4 0} C_DIS
LIN {X -37.289, Y 95.158, Z 165.75, A 0, B 90, C 0, E1 0, E2 0, E3 0, E4 0} C_DIS
LIN {X -34.383, Y 96.069, Z 165.75, A 0, B 90, C 0, E1 0, E2 0, E3 0, E4 0} C_DIS
LIN {X -31.404, Y 96.699, Z 165.75, A 0, B 90, C 0, E1 0, E2 0, E3 0, E4 0} C_DIS
LIN {X -28.379, Y 97.048, Z 165.75, A 0, B 90, C 0, E1 0, E2 0, E3 0, E4 0} C_DIS
LIN {X -25.334, Y 97.122, Z 165.75, A 0, B 90, C 0, E1 0, E2 0, E3 0, E4 0} C_DIS
LIN {X -22.295, Y 96.93, Z 165.75, A 0, B 90, C 0, E1 0, E2 0, E3 0, E4 0} C_DIS
LIN {X -19.282, Y 96.484, Z 165.75, A 0, B 90, C 0, E1 0, E2 0, E3 0, E4 0} C_DIS
LIN {X -16.315, Y 95.799, Z 165.75, A 0, B 90, C 0, E1 0, E2 0, E3 0, E4 0} C_DIS
LIN {X -13.407, Y 94.894, Z 165.75, A 0, B 90, C 0, E1 0, E2 0, E3 0, E4 0} C_DIS
LIN {X -10.568, Y 93.791, Z 165.75, A 0, B 90, C 0, E1 0, E2 0, E3 0, E4 0} C_DIS
LIN {X -7.801, Y 92.516, Z 165.75, A 0, B 90, C 0, E1 0, E2 0, E3 0, E4 0} C_DIS
LIN {X -5.107, Y 91.096, Z 165.75, A 0, B 90, C 0, E1 0, E2 0, E3 0, E4 0} C_DIS
LIN {X -2.487, Y 89.544, Z 165.75, A 0, B 90, C 0, E1 0, E2 0, E3 0, E4 0} C_DIS
LIN {X 0, Y 87.918, Z 165.75, A 0, B 90, C 0, E1 0, E2 0, E3 0, E4 0} C_DIS
LIN {X 2.051, Y 86.027, Z 165.75, A 0, B 90, C 0, E1 0, E2 0, E3 0, E4 0} C_DIS
LIN {X 4.479, Y 84.189, Z 165.75, A 0, B 90, C 0, E1 0, E2 0, E3 0, E4 0} C_DIS
LIN {X 6.882, Y 82.316, Z 165.75, A 0, B 90, C 0, E1 0, E2 0, E3 0, E4 0} C_DIS
LIN {X 9.252, Y 80.403, Z 165.75, A 0, B 90, C 0, E1 0, E2 0, E3 0, E4 0} C_DIS
LIN {X 11.614, Y 78.479, Z 165.75, A 0, B 90, C 0, E1 0, E2 0, E3 0, E4 0} C_DIS
LIN {X 13.994, Y 76.578, Z 165.75, A 0, B 90, C 0, E1 0, E2 0, E3 0, E4 0} C_DIS
LIN {X 16.416, Y 74.73, Z 165.75, A 0, B 90, C 0, E1 0, E2 0, E3 0, E4 0} C_DIS
LIN {X 18.897, Y 72.963, Z 165.75, A 0, B 90, C 0, E1 0, E2 0, E3 0, E4 0} C_DIS
LIN {X 21.457, Y 71.314, Z 165.75, A 0, B 90, C 0, E1 0, E2 0, E3 0, E4 0} C_DIS
LIN {X 24.118, Y 69.831, Z 165.75, A 0, B 90, C 0, E1 0, E2 0, E3 0, E4 0} C_DIS
LIN {X 26.885, Y 68.56, Z 165.75, A 0, B 90, C 0, E1 0, E2 0, E3 0, E4 0} C_DIS
LIN {X 29.753, Y 67.534, Z 165.75, A 0, B 90, C 0, E1 0, E2 0, E3 0, E4 0} C_DIS
LIN {X 32.695, Y 66.748, Z 165.75, A 0, B 90, C 0, E1 0, E2 0, E3 0, E4 0} C_DIS
LIN {X 35.686, Y 66.17, Z 165.75, A 0, B 90, C 0, E1 0, E2 0, E3 0, E4 0} C_DIS
LIN {X 38.702, Y 65.747, Z 165.75, A 0, B 90, C 0, E1 0, E2 0, E3 0, E4 0} C_DIS
LIN {X 41.731, Y 65.421, Z 165.75, A 0, B 90, C 0, E1 0, E2 0, E3 0, E4 0} C_DIS
LIN {X 44.764, Y 65.138, Z 165.75, A 0, B 90, C 0, E1 0, E2 0, E3 0, E4 0} C_DIS
LIN {X 47.797, Y 64.853, Z 165.75, A 0, B 90, C 0, E1 0, E2 0, E3 0, E4 0} C_DIS
LIN {X 50.826, Y 64.529, Z 165.75, A 0, B 90, C 0, E1 0, E2 0, E3 0, E4 0} C_DIS
LIN {X 53.847, Y 64.143, Z 165.75, A 0, B 90, C 0, E1 0, E2 0, E3 0, E4 0} C_DIS
LIN {X 56.858, Y 63.679, Z 165.75, A 0, B 90, C 0, E1 0, E2 0, E3 0, E4 0} C_DIS
LIN {X 59.853, Y 63.121, Z 165.75, A 0, B 90, C 0, E1 0, E2 0, E3 0, E4 0} C_DIS
LIN {X 62.826, Y 62.457, Z 165.75, A 0, B 90, C 0, E1 0, E2 0, E3 0, E4 0} C_DIS
LIN {X 65.769, Y 61.673, Z 165.75, A 0, B 90, C 0, E1 0, E2 0, E3 0, E4 0} C_DIS
LIN {X 68.673, Y 60.754, Z 165.75, A 0, B 90, C 0, E1 0, E2 0, E3 0, E4 0} C_DIS
LIN {X 71.527, Y 59.689, Z 165.75, A 0, B 90, C 0, E1 0, E2 0, E3 0, E4 0} C_DIS
LIN {X 74.317, Y 58.468, Z 165.75, A 0, B 90, C 0, E1 0, E2 0, E3 0, E4 0} C_DIS
LIN {X 77.029, Y 57.081, Z 165.75, A 0, B 90, C 0, E1 0, E2 0, E3 0, E4 0} C_DIS
LIN {X 79.646, Y 55.524, Z 165.75, A 0, B 90, C 0, E1 0, E2 0, E3 0, E4 0} C_DIS
LIN {X 82.155, Y 53.797, Z 165.75, A 0, B 90, C 0, E1 0, E2 0, E3 0, E4 0} C_DIS
LIN {X 84.547, Y 51.911, Z 165.75, A 0, B 90, C 0, E1 0, E2 0, E3 0, E4 0} C_DIS
LIN {X 86.808, Y 49.871, Z 165.75, A 0, B 90, C 0, E1 0, E2 0, E3 0, E4 0} C_DIS
LIN {X 88.913, Y 47.669, Z 165.75, A 0, B 90, C 0, E1 0, E2 0, E3 0, E4 0} C_DIS
LIN {X 90.827, Y 45.301, Z 165.75, A 0, B 90, C 0, E1 0, E2 0, E3 0, E4 0} C_DIS
LIN {X 92.521, Y 42.77, Z 165.75, A 0, B 90, C 0, E1 0, E2 0, E3 0, E4 0} C_DIS
LIN {X 93.971, Y 40.093, Z 165.75, A 0, B 90, C 0, E1 0, E2 0, E3 0, E4 0} C_DIS
LIN {X 95.158, Y 37.289, Z 165.75, A 0, B 90, C 0, E1 0, E2 0, E3 0, E4 0} C_DIS
LIN {X 96.069, Y 34.383, Z 165.75, A 0, B 90, C 0, E1 0, E2 0, E3 0, E4 0} C_DIS
LIN {X 96.699, Y 31.404, Z 165.75, A 0, B 90, C 0, E1 0, E2 0, E3 0, E4 0} C_DIS
LIN {X 97.048, Y 28.379, Z 165.75, A 0, B 90, C 0, E1 0, E2 0, E3 0, E4 0} C_DIS
LIN {X 97.122, Y 25.334, Z 165.75, A 0, B 90, C 0, E1 0, E2 0, E3 0, E4 0} C_DIS
LIN {X 96.93, Y 22.295, Z 165.75, A 0, B 90, C 0, E1 0, E2 0, E3 0, E4 0} C_DIS
LIN {X 96.484, Y 19.282, Z 165.75, A 0, B 90, C 0, E1 0, E2 0, E3 0, E4 0} C_DIS
LIN {X 95.799, Y 16.315, Z 165.75, A 0, B 90, C 0, E1 0, E2 0, E3 0, E4 0} C_DIS
LIN {X 94.894, Y 13.407, Z 165.75, A 0, B 90, C 0, E1 0, E2 0, E3 0, E4 0} C_DIS
LIN {X 93.791, Y 10.568, Z 165.75, A 0, B 90, C 0, E1 0, E2 0, E3 0, E4 0} C_DIS
LIN {X 92.516, Y 7.801, Z 165.75, A 0, B 90, C 0, E1 0, E2 0, E3 0, E4 0} C_DIS
LIN {X 91.096, Y 5.107, Z 165.75, A 0, B 90, C 0, E1 0, E2 0, E3 0, E4 0} C_DIS
LIN {X 89.544, Y 2.487, Z 165.75, A 0, B 90, C 0, E1 0, E2 0, E3 0, E4 0} C_DIS
LIN {X 87.918, Y 0, Z 165.75, A 0, B 90, C 0, E1 0, E2 0, E3 0, E4 0} C_DIS
LIN {X 86.027, Y -2.051, Z 165.75, A 0, B 90, C 0, E1 0, E2 0, E3 0, E4 0} C_DIS
LIN {X 84.189, Y -4.479, Z 165.75, A 0, B 90, C 0, E1 0, E2 0, E3 0, E4 0} C_DIS
LIN {X 82.316, Y -6.882, Z 165.75, A 0, B 90, C 0, E1 0, E2 0, E3 0, E4 0} C_DIS
LIN {X 80.403, Y -9.252, Z 165.75, A 0, B 90, C 0, E1 0, E2 0, E3 0, E4 0} C_DIS
LIN {X 78.479, Y -11.614, Z 165.75, A 0, B 90, C 0, E1 0, E2 0, E3 0, E4 0} C_DIS
LIN {X 76.578, Y -13.994, Z 165.75, A 0, B 90, C 0, E1 0, E2 0, E3 0, E4 0} C_DIS
LIN {X 74.73, Y -16.416, Z 165.75, A 0, B 90, C 0, E1 0, E2 0, E3 0, E4 0} C_DIS
LIN {X 72.963, Y -18.897, Z 165.75, A 0, B 90, C 0, E1 0, E2 0, E3 0, E4 0} C_DIS
LIN {X 71.314, Y -21.457, Z 165.75, A 0, B 90, C 0, E1 0, E2 0, E3 0, E4 0} C_DIS
LIN {X 69.831, Y -24.118, Z 165.75, A 0, B 90, C 0, E1 0, E2 0, E3 0, E4 0} C_DIS
LIN {X 68.56, Y -26.885, Z 165.75, A 0, B 90, C 0, E1 0, E2 0, E3 0, E4 0} C_DIS
LIN {X 67.534, Y -29.753, Z 165.75, A 0, B 90, C 0, E1 0, E2 0, E3 0, E4 0} C_DIS
LIN {X 66.748, Y -32.695, Z 165.75, A 0, B 90, C 0, E1 0, E2 0, E3 0, E4 0} C_DIS
LIN {X 66.17, Y -35.686, Z 165.75, A 0, B 90, C 0, E1 0, E2 0, E3 0, E4 0} C_DIS
LIN {X 65.747, Y -38.702, Z 165.75, A 0, B 90, C 0, E1 0, E2 0, E3 0, E4 0} C_DIS
LIN {X 65.421, Y -41.731, Z 165.75, A 0, B 90, C 0, E1 0, E2 0, E3 0, E4 0} C_DIS
LIN {X 65.138, Y -44.764, Z 165.75, A 0, B 90, C 0, E1 0, E2 0, E3 0, E4 0} C_DIS
LIN {X 64.853, Y -47.797, Z 165.75, A 0, B 90, C 0, E1 0, E2 0, E3 0, E4 0} C_DIS
LIN {X 64.529, Y -50.826, Z 165.75, A 0, B 90, C 0, E1 0, E2 0, E3 0, E4 0} C_DIS
LIN {X 64.143, Y -53.847, Z 165.75, A 0, B 90, C 0, E1 0, E2 0, E3 0, E4 0} C_DIS
LIN {X 63.679, Y -56.858, Z 165.75, A 0, B 90, C 0, E1 0, E2 0, E3 0, E4 0} C_DIS
LIN {X 63.121, Y -59.853, Z 165.75, A 0, B 90, C 0, E1 0, E2 0, E3 0, E4 0} C_DIS
LIN {X 62.457, Y -62.826, Z 165.75, A 0, B 90, C 0, E1 0, E2 0, E3 0, E4 0} C_DIS
LIN {X 61.673, Y -65.769, Z 165.75, A 0, B 90, C 0, E1 0, E2 0, E3 0, E4 0} C_DIS
LIN {X 60.754, Y -68.673, Z 165.75, A 0, B 90, C 0, E1 0, E2 0, E3 0, E4 0} C_DIS
LIN {X 59.689, Y -71.527, Z 165.75, A 0, B 90, C 0, E1 0, E2 0, E3 0, E4 0} C_DIS
LIN {X 58.468, Y -74.317, Z 165.75, A 0, B 90, C 0, E1 0, E2 0, E3 0, E4 0} C_DIS
LIN {X 57.081, Y -77.029, Z 165.75, A 0, B 90, C 0, E1 0, E2 0, E3 0, E4 0} C_DIS
LIN {X 55.524, Y -79.646, Z 165.75, A 0, B 90, C 0, E1 0, E2 0, E3 0, E4 0} C_DIS
LIN {X 53.797, Y -82.155, Z 165.75, A 0, B 90, C 0, E1 0, E2 0, E3 0, E4 0} C_DIS
LIN {X 51.911, Y -84.547, Z 165.75, A 0, B 90, C 0, E1 0, E2 0, E3 0, E4 0} C_DIS
LIN {X 49.871, Y -86.808, Z 165.75, A 0, B 90, C 0, E1 0, E2 0, E3 0, E4 0} C_DIS
LIN {X 47.669, Y -88.913, Z 165.75, A 0, B 90, C 0, E1 0, E2 0, E3 0, E4 0} C_DIS
LIN {X 45.301, Y -90.827, Z 165.75, A 0, B 90, C 0, E1 0, E2 0, E3 0, E4 0} C_DIS
LIN {X 42.77, Y -92.521, Z 165.75, A 0, B 90, C 0, E1 0, E2 0, E3 0, E4 0} C_DIS
LIN {X 40.093, Y -93.971, Z 165.75, A 0, B 90, C 0, E1 0, E2 0, E3 0, E4 0} C_DIS
LIN {X 37.289, Y -95.158, Z 165.75, A 0, B 90, C 0, E1 0, E2 0, E3 0, E4 0} C_DIS
LIN {X 34.383, Y -96.069, Z 165.75, A 0, B 90, C 0, E1 0, E2 0, E3 0, E4 0} C_DIS
LIN {X 31.404, Y -96.699, Z 165.75, A 0, B 90, C 0, E1 0, E2 0, E3 0, E4 0} C_DIS
LIN {X 28.379, Y -97.048, Z 165.75, A 0, B 90, C 0, E1 0, E2 0, E3 0, E4 0} C_DIS
LIN {X 25.334, Y -97.122, Z 165.75, A 0, B 90, C 0, E1 0, E2 0, E3 0, E4 0} C_DIS
LIN {X 22.295, Y -96.93, Z 165.75, A 0, B 90, C 0, E1 0, E2 0, E3 0, E4 0} C_DIS
LIN {X 19.282, Y -96.484, Z 165.75, A 0, B 90, C 0, E1 0, E2 0, E3 0, E4 0} C_DIS
LIN {X 16.315, Y -95.799, Z 165.75, A 0, B 90, C 0, E1 0, E2 0, E3 0, E4 0} C_DIS
LIN {X 13.407, Y -94.894, Z 165.75, A 0, B 90, C 0, E1 0, E2 0, E3 0, E4 0} C_DIS
LIN {X 10.568, Y -93.791, Z 165.75, A 0, B 90, C 0, E1 0, E2 0, E3 0, E4 0} C_DIS
LIN {X 7.801, Y -92.516, Z 165.75, A 0, B 90, C 0, E1 0, E2 0, E3 0, E4 0} C_DIS
LIN {X 5.107, Y -91.096, Z 165.75, A 0, B 90, C 0, E1 0, E2 0, E3 0, E4 0} C_DIS
LIN {X 2.487, Y -89.544, Z 165.75, A 0, B 90, C 0, E1 0, E2 0, E3 0, E4 0} C_DIS
LIN {X 0, Y -87.918, Z 165.75, A 0, B 90, C 0, E1 0, E2 0, E3 0, E4 0} C_DIS
LIN {X -2.051, Y -86.027, Z 165.75, A 0, B 90, C 0, E1 0, E2 0, E3 0, E4 0} C_DIS
LIN {X -4.479, Y -84.189, Z 165.75, A 0, B 90, C 0, E1 0, E2 0, E3 0, E4 0} C_DIS
LIN {X -6.882, Y -82.316, Z 165.75, A 0, B 90, C 0, E1 0, E2 0, E3 0, E4 0} C_DIS
LIN {X -9.252, Y -80.403, Z 165.75, A 0, B 90, C 0, E1 0, E2 0, E3 0, E4 0} C_DIS
LIN {X -11.614, Y -78.479, Z 165.75, A 0, B 90, C 0, E1 0, E2 0, E3 0, E4 0} C_DIS
LIN {X -13.994, Y -76.578, Z 165.75, A 0, B 90, C 0, E1 0, E2 0, E3 0, E4 0} C_DIS
LIN {X -16.416, Y -74.73, Z 165.75, A 0, B 90, C 0, E1 0, E2 0, E3 0, E4 0} C_DIS
LIN {X -18.897, Y -72.963, Z 165.75, A 0, B 90, C 0, E1 0, E2 0, E3 0, E4 0} C_DIS
LIN {X -21.457, Y -71.314, Z 165.75, A 0, B 90, C 0, E1 0, E2 0, E3 0, E4 0} C_DIS
LIN {X -24.118, Y -69.831, Z 165.75, A 0, B 90, C 0, E1 0, E2 0, E3 0, E4 0} C_DIS
LIN {X -26.885, Y -68.56, Z 165.75, A 0, B 90, C 0, E1 0, E2 0, E3 0, E4 0} C_DIS
LIN {X -29.753, Y -67.534, Z 165.75, A 0, B 90, C 0, E1 0, E2 0, E3 0, E4 0} C_DIS
LIN {X -32.695, Y -66.748, Z 165.75, A 0, B 90, C 0, E1 0, E2 0, E3 0, E4 0} C_DIS
LIN {X -35.686, Y -66.17, Z 165.75, A 0, B 90, C 0, E1 0, E2 0, E3 0, E4 0} C_DIS
LIN {X -38.702, Y -65.747, Z 165.75, A 0, B 90, C 0, E1 0, E2 0, E3 0, E4 0} C_DIS
LIN {X -41.731, Y -65.421, Z 165.75, A 0, B 90, C 0, E1 0, E2 0, E3 0, E4 0} C_DIS
LIN {X -44.764, Y -65.138, Z 165.75, A 0, B 90, C 0, E1 0, E2 0, E3 0, E4 0} C_DIS
LIN {X -47.797, Y -64.853, Z 165.75, A 0, B 90, C 0, E1 0, E2 0, E3 0, E4 0} C_DIS
LIN {X -50.826, Y -64.529, Z 165.75, A 0, B 90, C 0, E1 0, E2 0, E3 0, E4 0} C_DIS
LIN {X -53.847, Y -64.143, Z 165.75, A 0, B 90, C 0, E1 0, E2 0, E3 0, E4 0} C_DIS
LIN {X -56.858, Y -63.679, Z 165.75, A 0, B 90, C 0, E1 0, E2 0, E3 0, E4 0} C_DIS
LIN {X -59.853, Y -63.121, Z 165.75, A 0, B 90, C 0, E1 0, E2 0, E3 0, E4 0} C_DIS
LIN {X -62.826, Y -62.457, Z 165.75, A 0, B 90, C 0, E1 0, E2 0, E3 0, E4 0} C_DIS
LIN {X -65.769, Y -61.673, Z 165.75, A 0, B 90, C 0, E1 0, E2 0, E3 0, E4 0} C_DIS
LIN {X -68.673, Y -60.754, Z 165.75, A 0, B 90, C 0, E1 0, E2 0, E3 0, E4 0} C_DIS
LIN {X -71.527, Y -59.689, Z 165.75, A 0, B 90, C 0, E1 0, E2 0, E3 0, E4 0} C_DIS
LIN {X -74.317, Y -58.468, Z 165.75, A 0, B 90, C 0, E1 0, E2 0, E3 0, E4 0} C_DIS
LIN {X -77.029, Y -57.081, Z 165.75, A 0, B 90, C 0, E1 0, E2 0, E3 0, E4 0} C_DIS
LIN {X -79.646, Y -55.524, Z 165.75, A 0, B 90, C 0, E1 0, E2 0, E3 0, E4 0} C_DIS
LIN {X -82.155, Y -53.797, Z 165.75, A 0, B 90, C 0, E1 0, E2 0, E3 0, E4 0} C_DIS
LIN {X -84.547, Y -51.911, Z 165.75, A 0, B 90, C 0, E1 0, E2 0, E3 0, E4 0} C_DIS
LIN {X -86.808, Y -49.871, Z 165.75, A 0, B 90, C 0, E1 0, E2 0, E3 0, E4 0} C_DIS
LIN {X -88.913, Y -47.669, Z 165.75, A 0, B 90, C 0, E1 0, E2 0, E3 0, E4 0} C_DIS
LIN {X -90.827, Y -45.301, Z 165.75, A 0, B 90, C 0, E1 0, E2 0, E3 0, E4 0} C_DIS
LIN {X -92.521, Y -42.77, Z 165.75, A 0, B 90, C 0, E1 0, E2 0, E3 0, E4 0} C_DIS
LIN {X -93.971, Y -40.093, Z 165.75, A 0, B 90, C 0, E1 0, E2 0, E3 0, E4 0} C_DIS
LIN {X -95.158, Y -37.289, Z 165.75, A 0, B 90, C 0, E1 0, E2 0, E3 0, E4 0} C_DIS
LIN {X -96.069, Y -34.383, Z 165.75, A 0, B 90, C 0, E1 0, E2 0, E3 0, E4 0} C_DIS
LIN {X -96.699, Y -31.404, Z 165.75, A 0, B 90, C 0, E1 0, E2 0, E3 0, E4 0} C_DIS
LIN {X -97.048, Y -28.379, Z 165.75, A 0, B 90, C 0, E1 0, E2 0, E3 0, E4 0} C_DIS
LIN {X -97.122, Y -25.334, Z 165.75, A 0, B 90, C 0, E1 0, E2 0, E3 0, E4 0} C_DIS
LIN {X -96.93, Y -22.295, Z 165.75, A 0, B 90, C 0, E1 0, E2 0, E3 0, E4 0} C_DIS
LIN {X -96.484, Y -19.282, Z 165.75, A 0, B 90, C 0, E1 0, E2 0, E3 0, E4 0} C_DIS
LIN {X -95.799, Y -16.315, Z 165.75, A 0, B 90, C 0, E1 0, E2 0, E3 0, E4 0} C_DIS
LIN {X -94.894, Y -13.407, Z 165.75, A 0, B 90, C 0, E1 0, E2 0, E3 0, E4 0} C_DIS
LIN {X -93.791, Y -10.568, Z 165.75, A 0, B 90, C 0, E1 0, E2 0, E3 0, E4 0} C_DIS
LIN {X -92.516, Y -7.801, Z 165.75, A 0, B 90, C 0, E1 0, E2 0, E3 0, E4 0} C_DIS
LIN {X -91.096, Y -5.107, Z 165.75, A 0, B 90, C 0, E1 0, E2 0, E3 0, E4 0} C_DIS
LIN {X -89.544, Y -2.487, Z 165.75, A 0, B 90, C 0, E1 0, E2 0, E3 0, E4 0} C_DIS
LIN {X -88.338, Y 0, Z 168.25, A 0, B 90, C 0, E1 0, E2 0, E3 0, E4 0} C_DIS
LIN {X -86.428, Y 2.048, Z 168.25, A 0, B 90, C 0, E1 0, E2 0, E3 0, E4 0} C_DIS
LIN {X -84.569, Y 4.476, Z 168.25, A 0, B 90, C 0, E1 0, E2 0, E3 0, E4 0} C_DIS
LIN {X -82.677, Y 6.879, Z 168.25, A 0, B 90, C 0, E1 0, E2 0, E3 0, E4 0} C_DIS
LIN {X -80.748, Y 9.253, Z 168.25, A 0, B 90, C 0, E1 0, E2 0, E3 0, E4 0} C_DIS
LIN {X -78.812, Y 11.62, Z 168.25, A 0, B 90, C 0, E1 0, E2 0, E3 0, E4 0} C_DIS
LIN {X -76.908, Y 14.014, Z 168.25, A 0, B 90, C 0, E1 0, E2 0, E3 0, E4 0} C_DIS
LIN {X -75.068, Y 16.457, Z 168.25, A 0, B 90, C 0, E1 0, E2 0, E3 0, E4 0} C_DIS
LIN {X -73.316, Y 18.965, Z 168.25, A 0, B 90, C 0, E1 0, E2 0, E3 0, E4 0} C_DIS
LIN {X -71.687, Y 21.553, Z 168.25, A 0, B 90, C 0, E1 0, E2 0, E3 0, E4 0} C_DIS
LIN {X -70.226, Y 24.24, Z 168.25, A 0, B 90, C 0, E1 0, E2 0, E3 0, E4 0} C_DIS
LIN {X -68.981, Y 27.032, Z 168.25, A 0, B 90, C 0, E1 0, E2 0, E3 0, E4 0} C_DIS
LIN {X -67.98, Y 29.922, Z 168.25, A 0, B 90, C 0, E1 0, E2 0, E3 0, E4 0} C_DIS
LIN {X -67.22, Y 32.883, Z 168.25, A 0, B 90, C 0, E1 0, E2 0, E3 0, E4 0} C_DIS
LIN {X -66.665, Y 35.891, Z 168.25, A 0, B 90, C 0, E1 0, E2 0, E3 0, E4 0} C_DIS
LIN {X -66.261, Y 38.923, Z 168.25, A 0, B 90, C 0, E1 0, E2 0, E3 0, E4 0} C_DIS
LIN {X -65.949, Y 41.965, Z 168.25, A 0, B 90, C 0, E1 0, E2 0, E3 0, E4 0} C_DIS
LIN {X -65.673, Y 45.012, Z 168.25, A 0, B 90, C 0, E1 0, E2 0, E3 0, E4 0} C_DIS
LIN {X -65.385, Y 48.057, Z 168.25, A 0, B 90, C 0, E1 0, E2 0, E3 0, E4 0} C_DIS
LIN {X -65.048, Y 51.097, Z 168.25, A 0, B 90, C 0, E1 0, E2 0, E3 0, E4 0} C_DIS
LIN {X -64.64, Y 54.128, Z 168.25, A 0, B 90, C 0, E1 0, E2 0, E3 0, E4 0} C_DIS
LIN {X -64.145, Y 57.146, Z 168.25, A 0, B 90, C 0, E1 0, E2 0, E3 0, E4 0} C_DIS
LIN {X -63.554, Y 60.147, Z 168.25, A 0, B 90, C 0, E1 0, E2 0, E3 0, E4 0} C_DIS
LIN {X -62.853, Y 63.124, Z 168.25, A 0, B 90, C 0, E1 0, E2 0, E3 0, E4 0} C_DIS
LIN {X -62.029, Y 66.07, Z 168.25, A 0, B 90, C 0, E1 0, E2 0, E3 0, E4 0} C_DIS
LIN {X -61.07, Y 68.974, Z 168.25, A 0, B 90, C 0, E1 0, E2 0, E3 0, E4 0} C_DIS
LIN {X -59.964, Y 71.825, Z 168.25, A 0, B 90, C 0, E1 0, E2 0, E3 0, E4 0} C_DIS
LIN {X -58.7, Y 74.61, Z 168.25, A 0, B 90, C 0, E1 0, E2 0, E3 0, E4 0} C_DIS
LIN {X -57.271, Y 77.314, Z 168.25, A 0, B 90, C 0, E1 0, E2 0, E3 0, E4 0} C_DIS
LIN {X -55.673, Y 79.921, Z 168.25, A 0, B 90, C 0, E1 0, E2 0, E3 0, E4 0} C_DIS
LIN {X -53.912, Y 82.422, Z 168.25, A 0, B 90, C 0, E1 0, E2 0, E3 0, E4 0} C_DIS
LIN {X -52.004, Y 84.811, Z 168.25, A 0, B 90, C 0, E1 0, E2 0, E3 0, E4 0} C_DIS
LIN {X -49.955, Y 87.082, Z 168.25, A 0, B 90, C 0, E1 0, E2 0, E3 0, E4 0} C_DIS
LIN {X -47.754, Y 89.204, Z 168.25, A 0, B 90, C 0, E1 0, E2 0, E3 0, E4 0} C_DIS
LIN {X -45.388, Y 91.142, Z 168.25, A 0, B 90, C 0, E1 0, E2 0, E3 0, E4 0} C_DIS
LIN {X -42.862, Y 92.865, Z 168.25, A 0, B 90, C 0, E1 0, E2 0, E3 0, E4 0} C_DIS
LIN {X -40.186, Y 94.344, Z 168.25, A 0, B 90, C 0, E1 0, E2 0, E3 0, E4 0} C_DIS
LIN {X -37.382, Y 95.562, Z 168.25, A 0, B 90, C 0, E1 0, E2 0, E3 0, E4 0} C_DIS
LIN {X -34.473, Y 96.504, Z 168.25, A 0, B 90, C 0, E1 0, E2 0, E3 0, E4 0} C_DIS
LIN {X -31.487, Y 97.162, Z 168.25, A 0, B 90, C 0, E1 0, E2 0, E3 0, E4 0} C_DIS
LIN {X -28.453, Y 97.536, Z 168.25, A 0, B 90, C 0, E1 0, E2 0, E3 0, E4 0} C_DIS
LIN {X -25.396, Y 97.632, Z 168.25, A 0, B 90, C 0, E1 0, E2 0, E3 0, E4 0} C_DIS
LIN {X -22.344, Y 97.456, Z 168.25, A 0, B 90, C 0, E1 0, E2 0, E3 0, E4 0} C_DIS
LIN {X -19.318, Y 97.018, Z 168.25, A 0, B 90, C 0, E1 0, E2 0, E3 0, E4 0} C_DIS
LIN {X -16.338, Y 96.332, Z 168.25, A 0, B 90, C 0, E1 0, E2 0, E3 0, E4 0} C_DIS
LIN {X -13.42, Y 95.417, Z 168.25, A 0, B 90, C 0, E1 0, E2 0, E3 0, E4 0} C_DIS
LIN {X -10.574, Y 94.298, Z 168.25, A 0, B 90, C 0, E1 0, E2 0, E3 0, E4 0} C_DIS
LIN {X -7.803, Y 93.003, Z 168.25, A 0, B 90, C 0, E1 0, E2 0, E3 0, E4 0} C_DIS
LIN {X -5.106, Y 91.561, Z 168.25, A 0, B 90, C 0, E1 0, E2 0, E3 0, E4 0} C_DIS
LIN {X -2.486, Y 89.985, Z 168.25, A 0, B 90, C 0, E1 0, E2 0, E3 0, E4 0} C_DIS
LIN {X 0, Y 88.338, Z 168.25, A 0, B 90, C 0, E1 0, E2 0, E3 0, E4 0} C_DIS
LIN {X 2.048, Y 86.428, Z 168.25, A 0, B 90, C 0, E1 0, E2 0, E3 0, E4 0} C_DIS
LIN {X 4.476, Y 84.569, Z 168.25, A 0, B 90, C 0, E1 0, E2 0, E3 0, E4 0} C_DIS
LIN {X 6.879, Y 82.677, Z 168.25, A 0, B 90, C 0, E1 0, E2 0, E3 0, E4 0} C_DIS
LIN {X 9.253, Y 80.748, Z 168.25, A 0, B 90, C 0, E1 0, E2 0, E3 0, E4 0} C_DIS
LIN {X 11.62, Y 78.812, Z 168.25, A 0, B 90, C 0, E1 0, E2 0, E3 0, E4 0} C_DIS
LIN {X 14.014, Y 76.908, Z 168.25, A 0, B 90, C 0, E1 0, E2 0, E3 0, E4 0} C_DIS
LIN {X 16.457, Y 75.068, Z 168.25, A 0, B 90, C 0, E1 0, E2 0, E3 0, E4 0} C_DIS
LIN {X 18.965, Y 73.316, Z 168.25, A 0, B 90, C 0, E1 0, E2 0, E3 0, E4 0} C_DIS
LIN {X 21.553, Y 71.687, Z 168.25, A 0, B 90, C 0, E1 0, E2 0, E3 0, E4 0} C_DIS
LIN {X 24.24, Y 70.226, Z 168.25, A 0, B 90, C 0, E1 0, E2 0, E3 0, E4 0} C_DIS
LIN {X 27.032, Y 68.981, Z 168.25, A 0, B 90, C 0, E1 0, E2 0, E3 0, E4 0} C_DIS
LIN {X 29.922, Y 67.98, Z 168.25, A 0, B 90, C 0, E1 0, E2 0, E3 0, E4 0} C_DIS
LIN {X 32.883, Y 67.22, Z 168.25, A 0, B 90, C 0, E1 0, E2 0, E3 0, E4 0} C_DIS
LIN {X 35.891, Y 66.665, Z 168.25, A 0, B 90, C 0, E1 0, E2 0, E3 0, E4 0} C_DIS
LIN {X 38.923, Y 66.261, Z 168.25, A 0, B 90, C 0, E1 0, E2 0, E3 0, E4 0} C_DIS
LIN {X 41.965, Y 65.949, Z 168.25, A 0, B 90, C 0, E1 0, E2 0, E3 0, E4 0} C_DIS
LIN {X 45.012, Y 65.673, Z 168.25, A 0, B 90, C 0, E1 0, E2 0, E3 0, E4 0} C_DIS
LIN {X 48.057, Y 65.385, Z 168.25, A 0, B 90, C 0, E1 0, E2 0, E3 0, E4 0} C_DIS
LIN {X 51.097, Y 65.048, Z 168.25, A 0, B 90, C 0, E1 0, E2 0, E3 0, E4 0} C_DIS
LIN {X 54.128, Y 64.64, Z 168.25, A 0, B 90, C 0, E1 0, E2 0, E3 0, E4 0} C_DIS
LIN {X 57.146, Y 64.145, Z 168.25, A 0, B 90, C 0, E1 0, E2 0, E3 0, E4 0} C_DIS
LIN {X 60.147, Y 63.554, Z 168.25, A 0, B 90, C 0, E1 0, E2 0, E3 0, E4 0} C_DIS
LIN {X 63.124, Y 62.853, Z 168.25, A 0, B 90, C 0, E1 0, E2 0, E3 0, E4 0} C_DIS
LIN {X 66.07, Y 62.029, Z 168.25, A 0, B 90, C 0, E1 0, E2 0, E3 0, E4 0} C_DIS
LIN {X 68.974, Y 61.07, Z 168.25, A 0, B 90, C 0, E1 0, E2 0, E3 0, E4 0} C_DIS
LIN {X 71.825, Y 59.964, Z 168.25, A 0, B 90, C 0, E1 0, E2 0, E3 0, E4 0} C_DIS
LIN {X 74.61, Y 58.7, Z 168.25, A 0, B 90, C 0, E1 0, E2 0, E3 0, E4 0} C_DIS
LIN {X 77.314, Y 57.271, Z 168.25, A 0, B 90, C 0, E1 0, E2 0, E3 0, E4 0} C_DIS
LIN {X 79.921, Y 55.673, Z 168.25, A 0, B 90, C 0, E1 0, E2 0, E3 0, E4 0} C_DIS
LIN {X 82.422, Y 53.912, Z 168.25, A 0, B 90, C 0, E1 0, E2 0, E3 0, E4 0} C_DIS
LIN {X 84.811, Y 52.004, Z 168.25, A 0, B 90, C 0, E1 0, E2 0, E3 0, E4 0} C_DIS
LIN {X 87.082, Y 49.955, Z 168.25, A 0, B 90, C 0, E1 0, E2 0, E3 0, E4 0} C_DIS
LIN {X 89.204, Y 47.754, Z 168.25, A 0, B 90, C 0, E1 0, E2 0, E3 0, E4 0} C_DIS
LIN {X 91.142, Y 45.388, Z 168.25, A 0, B 90, C 0, E1 0, E2 0, E3 0, E4 0} C_DIS
LIN {X 92.865, Y 42.862, Z 168.25, A 0, B 90, C 0, E1 0, E2 0, E3 0, E4 0} C_DIS
LIN {X 94.344, Y 40.186, Z 168.25, A 0, B 90, C 0, E1 0, E2 0, E3 0, E4 0} C_DIS
LIN {X 95.562, Y 37.382, Z 168.25, A 0, B 90, C 0, E1 0, E2 0, E3 0, E4 0} C_DIS
LIN {X 96.504, Y 34.473, Z 168.25, A 0, B 90, C 0, E1 0, E2 0, E3 0, E4 0} C_DIS
LIN {X 97.162, Y 31.487, Z 168.25, A 0, B 90, C 0, E1 0, E2 0, E3 0, E4 0} C_DIS
LIN {X 97.536, Y 28.453, Z 168.25, A 0, B 90, C 0, E1 0, E2 0, E3 0, E4 0} C_DIS
LIN {X 97.632, Y 25.396, Z 168.25, A 0, B 90, C 0, E1 0, E2 0, E3 0, E4 0} C_DIS
LIN {X 97.456, Y 22.344, Z 168.25, A 0, B 90, C 0, E1 0, E2 0, E3 0, E4 0} C_DIS
LIN {X 97.018, Y 19.318, Z 168.25, A 0, B 90, C 0, E1 0, E2 0, E3 0, E4 0} C_DIS
LIN {X 96.332, Y 16.338, Z 168.25, A 0, B 90, C 0, E1 0, E2 0, E3 0, E4 0} C_DIS
LIN {X 95.417, Y 13.42, Z 168.25, A 0, B 90, C 0, E1 0, E2 0, E3 0, E4 0} C_DIS
LIN {X 94.298, Y 10.574, Z 168.25, A 0, B 90, C 0, E1 0, E2 0, E3 0, E4 0} C_DIS
LIN {X 93.003, Y 7.803, Z 168.25, A 0, B 90, C 0, E1 0, E2 0, E3 0, E4 0} C_DIS
LIN {X 91.561, Y 5.106, Z 168.25, A 0, B 90, C 0, E1 0, E2 0, E3 0, E4 0} C_DIS
LIN {X 89.985, Y 2.486, Z 168.25, A 0, B 90, C 0, E1 0, E2 0, E3 0, E4 0} C_DIS
LIN {X 88.338, Y 0, Z 168.25, A 0, B 90, C 0, E1 0, E2 0, E3 0, E4 0} C_DIS
LIN {X 86.428, Y -2.048, Z 168.25, A 0, B 90, C 0, E1 0, E2 0, E3 0, E4 0} C_DIS
LIN {X 84.569, Y -4.476, Z 168.25, A 0, B 90, C 0, E1 0, E2 0, E3 0, E4 0} C_DIS
LIN {X 82.677, Y -6.879, Z 168.25, A 0, B 90, C 0, E1 0, E2 0, E3 0, E4 0} C_DIS
LIN {X 80.748, Y -9.253, Z 168.25, A 0, B 90, C 0, E1 0, E2 0, E3 0, E4 0} C_DIS
LIN {X 78.812, Y -11.62, Z 168.25, A 0, B 90, C 0, E1 0, E2 0, E3 0, E4 0} C_DIS
LIN {X 76.908, Y -14.014, Z 168.25, A 0, B 90, C 0, E1 0, E2 0, E3 0, E4 0} C_DIS
LIN {X 75.068, Y -16.457, Z 168.25, A 0, B 90, C 0, E1 0, E2 0, E3 0, E4 0} C_DIS
LIN {X 73.316, Y -18.965, Z 168.25, A 0, B 90, C 0, E1 0, E2 0, E3 0, E4 0} C_DIS
LIN {X 71.687, Y -21.553, Z 168.25, A 0, B 90, C 0, E1 0, E2 0, E3 0, E4 0} C_DIS
LIN {X 70.226, Y -24.24, Z 168.25, A 0, B 90, C 0, E1 0, E2 0, E3 0, E4 0} C_DIS
LIN {X 68.981, Y -27.032, Z 168.25, A 0, B 90, C 0, E1 0, E2 0, E3 0, E4 0} C_DIS
LIN {X 67.98, Y -29.922, Z 168.25, A 0, B 90, C 0, E1 0, E2 0, E3 0, E4 0} C_DIS
LIN {X 67.22, Y -32.883, Z 168.25, A 0, B 90, C 0, E1 0, E2 0, E3 0, E4 0} C_DIS
LIN {X 66.665, Y -35.891, Z 168.25, A 0, B 90, C 0, E1 0, E2 0, E3 0, E4 0} C_DIS
LIN {X 66.261, Y -38.923, Z 168.25, A 0, B 90, C 0, E1 0, E2 0, E3 0, E4 0} C_DIS
LIN {X 65.949, Y -41.965, Z 168.25, A 0, B 90, C 0, E1 0, E2 0, E3 0, E4 0} C_DIS
LIN {X 65.673, Y -45.012, Z 168.25, A 0, B 90, C 0, E1 0, E2 0, E3 0, E4 0} C_DIS
LIN {X 65.385, Y -48.057, Z 168.25, A 0, B 90, C 0, E1 0, E2 0, E3 0, E4 0} C_DIS
LIN {X 65.048, Y -51.097, Z 168.25, A 0, B 90, C 0, E1 0, E2 0, E3 0, E4 0} C_DIS
LIN {X 64.64, Y -54.128, Z 168.25, A 0, B 90, C 0, E1 0, E2 0, E3 0, E4 0} C_DIS
LIN {X 64.145, Y -57.146, Z 168.25, A 0, B 90, C 0, E1 0, E2 0, E3 0, E4 0} C_DIS
LIN {X 63.554, Y -60.147, Z 168.25, A 0, B 90, C 0, E1 0, E2 0, E3 0, E4 0} C_DIS
LIN {X 62.853, Y -63.124, Z 168.25, A 0, B 90, C 0, E1 0, E2 0, E3 0, E4 0} C_DIS
LIN {X 62.029, Y -66.07, Z 168.25, A 0, B 90, C 0, E1 0, E2 0, E3 0, E4 0} C_DIS
LIN {X 61.07, Y -68.974, Z 168.25, A 0, B 90, C 0, E1 0, E2 0, E3 0, E4 0} C_DIS
LIN {X 59.964, Y -71.825, Z 168.25, A 0, B 90, C 0, E1 0, E2 0, E3 0, E4 0} C_DIS
LIN {X 58.7, Y -74.61, Z 168.25, A 0, B 90, C 0, E1 0, E2 0, E3 0, E4 0} C_DIS
LIN {X 57.271, Y -77.314, Z 168.25, A 0, B 90, C 0, E1 0, E2 0, E3 0, E4 0} C_DIS
LIN {X 55.673, Y -79.921, Z 168.25, A 0, B 90, C 0, E1 0, E2 0, E3 0, E4 0} C_DIS
LIN {X 53.912, Y -82.422, Z 168.25, A 0, B 90, C 0, E1 0, E2 0, E3 0, E4 0} C_DIS
LIN {X 52.004, Y -84.811, Z 168.25, A 0, B 90, C 0, E1 0, E2 0, E3 0, E4 0} C_DIS
LIN {X 49.955, Y -87.082, Z 168.25, A 0, B 90, C 0, E1 0, E2 0, E3 0, E4 0} C_DIS
LIN {X 47.754, Y -89.204, Z 168.25, A 0, B 90, C 0, E1 0, E2 0, E3 0, E4 0} C_DIS
LIN {X 45.388, Y -91.142, Z 168.25, A 0, B 90, C 0, E1 0, E2 0, E3 0, E4 0} C_DIS
LIN {X 42.862, Y -92.865, Z 168.25, A 0, B 90, C 0, E1 0, E2 0, E3 0, E4 0} C_DIS
LIN {X 40.186, Y -94.344, Z 168.25, A 0, B 90, C 0, E1 0, E2 0, E3 0, E4 0} C_DIS
LIN {X 37.382, Y -95.562, Z 168.25, A 0, B 90, C 0, E1 0, E2 0, E3 0, E4 0} C_DIS
LIN {X 34.473, Y -96.504, Z 168.25, A 0, B 90, C 0, E1 0, E2 0, E3 0, E4 0} C_DIS
LIN {X 31.487, Y -97.162, Z 168.25, A 0, B 90, C 0, E1 0, E2 0, E3 0, E4 0} C_DIS
LIN {X 28.453, Y -97.536, Z 168.25, A 0, B 90, C 0, E1 0, E2 0, E3 0, E4 0} C_DIS
LIN {X 25.396, Y -97.632, Z 168.25, A 0, B 90, C 0, E1 0, E2 0, E3 0, E4 0} C_DIS
LIN {X 22.344, Y -97.456, Z 168.25, A 0, B 90, C 0, E1 0, E2 0, E3 0, E4 0} C_DIS
LIN {X 19.318, Y -97.018, Z 168.25, A 0, B 90, C 0, E1 0, E2 0, E3 0, E4 0} C_DIS
LIN {X 16.338, Y -96.332, Z 168.25, A 0, B 90, C 0, E1 0, E2 0, E3 0, E4 0} C_DIS
LIN {X 13.42, Y -95.417, Z 168.25, A 0, B 90, C 0, E1 0, E2 0, E3 0, E4 0} C_DIS
LIN {X 10.574, Y -94.298, Z 168.25, A 0, B 90, C 0, E1 0, E2 0, E3 0, E4 0} C_DIS
LIN {X 7.803, Y -93.003, Z 168.25, A 0, B 90, C 0, E1 0, E2 0, E3 0, E4 0} C_DIS
LIN {X 5.106, Y -91.561, Z 168.25, A 0, B 90, C 0, E1 0, E2 0, E3 0, E4 0} C_DIS
LIN {X 2.486, Y -89.985, Z 168.25, A 0, B 90, C 0, E1 0, E2 0, E3 0, E4 0} C_DIS
LIN {X 0, Y -88.338, Z 168.25, A 0, B 90, C 0, E1 0, E2 0, E3 0, E4 0} C_DIS
LIN {X -2.048, Y -86.428, Z 168.25, A 0, B 90, C 0, E1 0, E2 0, E3 0, E4 0} C_DIS
LIN {X -4.476, Y -84.569, Z 168.25, A 0, B 90, C 0, E1 0, E2 0, E3 0, E4 0} C_DIS
LIN {X -6.879, Y -82.677, Z 168.25, A 0, B 90, C 0, E1 0, E2 0, E3 0, E4 0} C_DIS
LIN {X -9.253, Y -80.748, Z 168.25, A 0, B 90, C 0, E1 0, E2 0, E3 0, E4 0} C_DIS
LIN {X -11.62, Y -78.812, Z 168.25, A 0, B 90, C 0, E1 0, E2 0, E3 0, E4 0} C_DIS
LIN {X -14.014, Y -76.908, Z 168.25, A 0, B 90, C 0, E1 0, E2 0, E3 0, E4 0} C_DIS
LIN {X -16.457, Y -75.068, Z 168.25, A 0, B 90, C 0, E1 0, E2 0, E3 0, E4 0} C_DIS
LIN {X -18.965, Y -73.316, Z 168.25, A 0, B 90, C 0, E1 0, E2 0, E3 0, E4 0} C_DIS
LIN {X -21.553, Y -71.687, Z 168.25, A 0, B 90, C 0, E1 0, E2 0, E3 0, E4 0} C_DIS
LIN {X -24.24, Y -70.226, Z 168.25, A 0, B 90, C 0, E1 0, E2 0, E3 0, E4 0} C_DIS
LIN {X -27.032, Y -68.981, Z 168.25, A 0, B 90, C 0, E1 0, E2 0, E3 0, E4 0} C_DIS
LIN {X -29.922, Y -67.98, Z 168.25, A 0, B 90, C 0, E1 0, E2 0, E3 0, E4 0} C_DIS
LIN {X -32.883, Y -67.22, Z 168.25, A 0, B 90, C 0, E1 0, E2 0, E3 0, E4 0} C_DIS
LIN {X -35.891, Y -66.665, Z 168.25, A 0, B 90, C 0, E1 0, E2 0, E3 0, E4 0} C_DIS
LIN {X -38.923, Y -66.261, Z 168.25, A 0, B 90, C 0, E1 0, E2 0, E3 0, E4 0} C_DIS
LIN {X -41.965, Y -65.949, Z 168.25, A 0, B 90, C 0, E1 0, E2 0, E3 0, E4 0} C_DIS
LIN {X -45.012, Y -65.673, Z 168.25, A 0, B 90, C 0, E1 0, E2 0, E3 0, E4 0} C_DIS
LIN {X -48.057, Y -65.385, Z 168.25, A 0, B 90, C 0, E1 0, E2 0, E3 0, E4 0} C_DIS
LIN {X -51.097, Y -65.048, Z 168.25, A 0, B 90, C 0, E1 0, E2 0, E3 0, E4 0} C_DIS
LIN {X -54.128, Y -64.64, Z 168.25, A 0, B 90, C 0, E1 0, E2 0, E3 0, E4 0} C_DIS
LIN {X -57.146, Y -64.145, Z 168.25, A 0, B 90, C 0, E1 0, E2 0, E3 0, E4 0} C_DIS
LIN {X -60.147, Y -63.554, Z 168.25, A 0, B 90, C 0, E1 0, E2 0, E3 0, E4 0} C_DIS
LIN {X -63.124, Y -62.853, Z 168.25, A 0, B 90, C 0, E1 0, E2 0, E3 0, E4 0} C_DIS
LIN {X -66.07, Y -62.029, Z 168.25, A 0, B 90, C 0, E1 0, E2 0, E3 0, E4 0} C_DIS
LIN {X -68.974, Y -61.07, Z 168.25, A 0, B 90, C 0, E1 0, E2 0, E3 0, E4 0} C_DIS
LIN {X -71.825, Y -59.964, Z 168.25, A 0, B 90, C 0, E1 0, E2 0, E3 0, E4 0} C_DIS
LIN {X -74.61, Y -58.7, Z 168.25, A 0, B 90, C 0, E1 0, E2 0, E3 0, E4 0} C_DIS
LIN {X -77.314, Y -57.271, Z 168.25, A 0, B 90, C 0, E1 0, E2 0, E3 0, E4 0} C_DIS
LIN {X -79.921, Y -55.673, Z 168.25, A 0, B 90, C 0, E1 0, E2 0, E3 0, E4 0} C_DIS
LIN {X -82.422, Y -53.912, Z 168.25, A 0, B 90, C 0, E1 0, E2 0, E3 0, E4 0} C_DIS
LIN {X -84.811, Y -52.004, Z 168.25, A 0, B 90, C 0, E1 0, E2 0, E3 0, E4 0} C_DIS
LIN {X -87.082, Y -49.955, Z 168.25, A 0, B 90, C 0, E1 0, E2 0, E3 0, E4 0} C_DIS
LIN {X -89.204, Y -47.754, Z 168.25, A 0, B 90, C 0, E1 0, E2 0, E3 0, E4 0} C_DIS
LIN {X -91.142, Y -45.388, Z 168.25, A 0, B 90, C 0, E1 0, E2 0, E3 0, E4 0} C_DIS
LIN {X -92.865, Y -42.862, Z 168.25, A 0, B 90, C 0, E1 0, E2 0, E3 0, E4 0} C_DIS
LIN {X -94.344, Y -40.186, Z 168.25, A 0, B 90, C 0, E1 0, E2 0, E3 0, E4 0} C_DIS
LIN {X -95.562, Y -37.382, Z 168.25, A 0, B 90, C 0, E1 0, E2 0, E3 0, E4 0} C_DIS
LIN {X -96.504, Y -34.473, Z 168.25, A 0, B 90, C 0, E1 0, E2 0, E3 0, E4 0} C_DIS
LIN {X -97.162, Y -31.487, Z 168.25, A 0, B 90, C 0, E1 0, E2 0, E3 0, E4 0} C_DIS
LIN {X -97.536, Y -28.453, Z 168.25, A 0, B 90, C 0, E1 0, E2 0, E3 0, E4 0} C_DIS
LIN {X -97.632, Y -25.396, Z 168.25, A 0, B 90, C 0, E1 0, E2 0, E3 0, E4 0} C_DIS
LIN {X -97.456, Y -22.344, Z 168.25, A 0, B 90, C 0, E1 0, E2 0, E3 0, E4 0} C_DIS
LIN {X -97.018, Y -19.318, Z 168.25, A 0, B 90, C 0, E1 0, E2 0, E3 0, E4 0} C_DIS
LIN {X -96.332, Y -16.338, Z 168.25, A 0, B 90, C 0, E1 0, E2 0, E3 0, E4 0} C_DIS
LIN {X -95.417, Y -13.42, Z 168.25, A 0, B 90, C 0, E1 0, E2 0, E3 0, E4 0} C_DIS
LIN {X -94.298, Y -10.574, Z 168.25, A 0, B 90, C 0, E1 0, E2 0, E3 0, E4 0} C_DIS
LIN {X -93.003, Y -7.803, Z 168.25, A 0, B 90, C 0, E1 0, E2 0, E3 0, E4 0} C_DIS
LIN {X -91.561, Y -5.106, Z 168.25, A 0, B 90, C 0, E1 0, E2 0, E3 0, E4 0} C_DIS
LIN {X -89.985, Y -2.486, Z 168.25, A 0, B 90, C 0, E1 0, E2 0, E3 0, E4 0} C_DIS
LIN {X -88.767, Y 0, Z 170.75, A 0, B 90, C 0, E1 0, E2 0, E3 0, E4 0} C_DIS
LIN {X -86.839, Y 2.046, Z 170.75, A 0, B 90, C 0, E1 0, E2 0, E3 0, E4 0} C_DIS
LIN {X -84.959, Y 4.474, Z 170.75, A 0, B 90, C 0, E1 0, E2 0, E3 0, E4 0} C_DIS
LIN {X -83.048, Y 6.878, Z 170.75, A 0, B 90, C 0, E1 0, E2 0, E3 0, E4 0} C_DIS
LIN {X -81.102, Y 9.254, Z 170.75, A 0, B 90, C 0, E1 0, E2 0, E3 0, E4 0} C_DIS
LIN {X -79.154, Y 11.629, Z 170.75, A 0, B 90, C 0, E1 0, E2 0, E3 0, E4 0} C_DIS
LIN {X -77.247, Y 14.037, Z 170.75, A 0, B 90, C 0, E1 0, E2 0, E3 0, E4 0} C_DIS
LIN {X -75.416, Y 16.502, Z 170.75, A 0, B 90, C 0, E1 0, E2 0, E3 0, E4 0} C_DIS
LIN {X -73.681, Y 19.036, Z 170.75, A 0, B 90, C 0, E1 0, E2 0, E3 0, E4 0} C_DIS
LIN {X -72.073, Y 21.652, Z 170.75, A 0, B 90, C 0, E1 0, E2 0, E3 0, E4 0} C_DIS
LIN {X -70.637, Y 24.367, Z 170.75, A 0, B 90, C 0, E1 0, E2 0, E3 0, E4 0} C_DIS
LIN {X -69.417, Y 27.184, Z 170.75, A 0, B 90, C 0, E1 0, E2 0, E3 0, E4 0} C_DIS
LIN {X -68.444, Y 30.097, Z 170.75, A 0, B 90, C 0, E1 0, E2 0, E3 0, E4 0} C_DIS
LIN {X -67.71, Y 33.078, Z 170.75, A 0, B 90, C 0, E1 0, E2 0, E3 0, E4 0} C_DIS
LIN {X -67.179, Y 36.103, Z 170.75, A 0, B 90, C 0, E1 0, E2 0, E3 0, E4 0} C_DIS
LIN {X -66.795, Y 39.15, Z 170.75, A 0, B 90, C 0, E1 0, E2 0, E3 0, E4 0} C_DIS
LIN {X -66.497, Y 42.207, Z 170.75, A 0, B 90, C 0, E1 0, E2 0, E3 0, E4 0} C_DIS
LIN {X -66.228, Y 45.266, Z 170.75, A 0, B 90, C 0, E1 0, E2 0, E3 0, E4 0} C_DIS
LIN {X -65.937, Y 48.324, Z 170.75, A 0, B 90, C 0, E1 0, E2 0, E3 0, E4 0} C_DIS
LIN {X -65.586, Y 51.375, Z 170.75, A 0, B 90, C 0, E1 0, E2 0, E3 0, E4 0} C_DIS
LIN {X -65.154, Y 54.416, Z 170.75, A 0, B 90, C 0, E1 0, E2 0, E3 0, E4 0} C_DIS
LIN {X -64.628, Y 57.442, Z 170.75, A 0, B 90, C 0, E1 0, E2 0, E3 0, E4 0} C_DIS
LIN {X -64.001, Y 60.448, Z 170.75, A 0, B 90, C 0, E1 0, E2 0, E3 0, E4 0} C_DIS
LIN {X -63.261, Y 63.429, Z 170.75, A 0, B 90, C 0, E1 0, E2 0, E3 0, E4 0} C_DIS
LIN {X -62.396, Y 66.375, Z 170.75, A 0, B 90, C 0, E1 0, E2 0, E3 0, E4 0} C_DIS
LIN {X -61.394, Y 69.278, Z 170.75, A 0, B 90, C 0, E1 0, E2 0, E3 0, E4 0} C_DIS
LIN {X -60.243, Y 72.126, Z 170.75, A 0, B 90, C 0, E1 0, E2 0, E3 0, E4 0} C_DIS
LIN {X -58.935, Y 74.904, Z 170.75, A 0, B 90, C 0, E1 0, E2 0, E3 0, E4 0} C_DIS
LIN {X -57.462, Y 77.598, Z 170.75, A 0, B 90, C 0, E1 0, E2 0, E3 0, E4 0} C_DIS
LIN {X -55.823, Y 80.195, Z 170.75, A 0, B 90, C 0, E1 0, E2 0, E3 0, E4 0} C_DIS
LIN {X -54.027, Y 82.686, Z 170.75, A 0, B 90, C 0, E1 0, E2 0, E3 0, E4 0} C_DIS
LIN {X -52.096, Y 85.074, Z 170.75, A 0, B 90, C 0, E1 0, E2 0, E3 0, E4 0} C_DIS
LIN {X -50.039, Y 87.354, Z 170.75, A 0, B 90, C 0, E1 0, E2 0, E3 0, E4 0} C_DIS
LIN {X -47.838, Y 89.496, Z 170.75, A 0, B 90, C 0, E1 0, E2 0, E3 0, E4 0} C_DIS
LIN {X -45.476, Y 91.458, Z 170.75, A 0, B 90, C 0, E1 0, E2 0, E3 0, E4 0} C_DIS
LIN {X -42.954, Y 93.209, Z 170.75, A 0, B 90, C 0, E1 0, E2 0, E3 0, E4 0} C_DIS
LIN {X -40.281, Y 94.72, Z 170.75, A 0, B 90, C 0, E1 0, E2 0, E3 0, E4 0} C_DIS
LIN {X -37.477, Y 95.969, Z 170.75, A 0, B 90, C 0, E1 0, E2 0, E3 0, E4 0} C_DIS
LIN {X -34.565, Y 96.942, Z 170.75, A 0, B 90, C 0, E1 0, E2 0, E3 0, E4 0} C_DIS
LIN {X -31.573, Y 97.63, Z 170.75, A 0, B 90, C 0, E1 0, E2 0, E3 0, E4 0} C_DIS
LIN {X -28.529, Y 98.032, Z 170.75, A 0, B 90, C 0, E1 0, E2 0, E3 0, E4 0} C_DIS
LIN {X -25.461, Y 98.15, Z 170.75, A 0, B 90, C 0, E1 0, E2 0, E3 0, E4 0} C_DIS
LIN {X -22.395, Y 97.99, Z 170.75, A 0, B 90, C 0, E1 0, E2 0, E3 0, E4 0} C_DIS
LIN {X -19.355, Y 97.56, Z 170.75, A 0, B 90, C 0, E1 0, E2 0, E3 0, E4 0} C_DIS
LIN {X -16.362, Y 96.873, Z 170.75, A 0, B 90, C 0, E1 0, E2 0, E3 0, E4 0} C_DIS
LIN {X -13.434, Y 95.949, Z 170.75, A 0, B 90, C 0, E1 0, E2 0, E3 0, E4 0} C_DIS
LIN {X -10.58, Y 94.814, Z 170.75, A 0, B 90, C 0, E1 0, E2 0, E3 0, E4 0} C_DIS
LIN {X -7.805, Y 93.5, Z 170.75, A 0, B 90, C 0, E1 0, E2 0, E3 0, E4 0} C_DIS
LIN {X -5.106, Y 92.035, Z 170.75, A 0, B 90, C 0, E1 0, E2 0, E3 0, E4 0} C_DIS
LIN {X -2.485, Y 90.436, Z 170.75, A 0, B 90, C 0, E1 0, E2 0, E3 0, E4 0} C_DIS
LIN {X 0, Y 88.767, Z 170.75, A 0, B 90, C 0, E1 0, E2 0, E3 0, E4 0} C_DIS
LIN {X 2.046, Y 86.839, Z 170.75, A 0, B 90, C 0, E1 0, E2 0, E3 0, E4 0} C_DIS
LIN {X 4.474, Y 84.959, Z 170.75, A 0, B 90, C 0, E1 0, E2 0, E3 0, E4 0} C_DIS
LIN {X 6.878, Y 83.048, Z 170.75, A 0, B 90, C 0, E1 0, E2 0, E3 0, E4 0} C_DIS
LIN {X 9.254, Y 81.102, Z 170.75, A 0, B 90, C 0, E1 0, E2 0, E3 0, E4 0} C_DIS
LIN {X 11.629, Y 79.154, Z 170.75, A 0, B 90, C 0, E1 0, E2 0, E3 0, E4 0} C_DIS
LIN {X 14.037, Y 77.247, Z 170.75, A 0, B 90, C 0, E1 0, E2 0, E3 0, E4 0} C_DIS
LIN {X 16.502, Y 75.416, Z 170.75, A 0, B 90, C 0, E1 0, E2 0, E3 0, E4 0} C_DIS
LIN {X 19.036, Y 73.681, Z 170.75, A 0, B 90, C 0, E1 0, E2 0, E3 0, E4 0} C_DIS
LIN {X 21.652, Y 72.073, Z 170.75, A 0, B 90, C 0, E1 0, E2 0, E3 0, E4 0} C_DIS
LIN {X 24.367, Y 70.637, Z 170.75, A 0, B 90, C 0, E1 0, E2 0, E3 0, E4 0} C_DIS
LIN {X 27.184, Y 69.417, Z 170.75, A 0, B 90, C 0, E1 0, E2 0, E3 0, E4 0} C_DIS
LIN {X 30.097, Y 68.444, Z 170.75, A 0, B 90, C 0, E1 0, E2 0, E3 0, E4 0} C_DIS
LIN {X 33.078, Y 67.71, Z 170.75, A 0, B 90, C 0, E1 0, E2 0, E3 0, E4 0} C_DIS
LIN {X 36.103, Y 67.179, Z 170.75, A 0, B 90, C 0, E1 0, E2 0, E3 0, E4 0} C_DIS
LIN {X 39.15, Y 66.795, Z 170.75, A 0, B 90, C 0, E1 0, E2 0, E3 0, E4 0} C_DIS
LIN {X 42.207, Y 66.497, Z 170.75, A 0, B 90, C 0, E1 0, E2 0, E3 0, E4 0} C_DIS
LIN {X 45.266, Y 66.228, Z 170.75, A 0, B 90, C 0, E1 0, E2 0, E3 0, E4 0} C_DIS
LIN {X 48.324, Y 65.937, Z 170.75, A 0, B 90, C 0, E1 0, E2 0, E3 0, E4 0} C_DIS
LIN {X 51.375, Y 65.586, Z 170.75, A 0, B 90, C 0, E1 0, E2 0, E3 0, E4 0} C_DIS
LIN {X 54.416, Y 65.154, Z 170.75, A 0, B 90, C 0, E1 0, E2 0, E3 0, E4 0} C_DIS
LIN {X 57.442, Y 64.628, Z 170.75, A 0, B 90, C 0, E1 0, E2 0, E3 0, E4 0} C_DIS
LIN {X 60.448, Y 64.001, Z 170.75, A 0, B 90, C 0, E1 0, E2 0, E3 0, E4 0} C_DIS
LIN {X 63.429, Y 63.261, Z 170.75, A 0, B 90, C 0, E1 0, E2 0, E3 0, E4 0} C_DIS
LIN {X 66.375, Y 62.396, Z 170.75, A 0, B 90, C 0, E1 0, E2 0, E3 0, E4 0} C_DIS
LIN {X 69.278, Y 61.394, Z 170.75, A 0, B 90, C 0, E1 0, E2 0, E3 0, E4 0} C_DIS
LIN {X 72.126, Y 60.243, Z 170.75, A 0, B 90, C 0, E1 0, E2 0, E3 0, E4 0} C_DIS
LIN {X 74.904, Y 58.935, Z 170.75, A 0, B 90, C 0, E1 0, E2 0, E3 0, E4 0} C_DIS
LIN {X 77.598, Y 57.462, Z 170.75, A 0, B 90, C 0, E1 0, E2 0, E3 0, E4 0} C_DIS
LIN {X 80.195, Y 55.823, Z 170.75, A 0, B 90, C 0, E1 0, E2 0, E3 0, E4 0} C_DIS
LIN {X 82.686, Y 54.027, Z 170.75, A 0, B 90, C 0, E1 0, E2 0, E3 0, E4 0} C_DIS
LIN {X 85.074, Y 52.096, Z 170.75, A 0, B 90, C 0, E1 0, E2 0, E3 0, E4 0} C_DIS
LIN {X 87.354, Y 50.039, Z 170.75, A 0, B 90, C 0, E1 0, E2 0, E3 0, E4 0} C_DIS
LIN {X 89.496, Y 47.838, Z 170.75, A 0, B 90, C 0, E1 0, E2 0, E3 0, E4 0} C_DIS
LIN {X 91.458, Y 45.476, Z 170.75, A 0, B 90, C 0, E1 0, E2 0, E3 0, E4 0} C_DIS
LIN {X 93.209, Y 42.954, Z 170.75, A 0, B 90, C 0, E1 0, E2 0, E3 0, E4 0} C_DIS
LIN {X 94.72, Y 40.281, Z 170.75, A 0, B 90, C 0, E1 0, E2 0, E3 0, E4 0} C_DIS
LIN {X 95.969, Y 37.477, Z 170.75, A 0, B 90, C 0, E1 0, E2 0, E3 0, E4 0} C_DIS
LIN {X 96.942, Y 34.565, Z 170.75, A 0, B 90, C 0, E1 0, E2 0, E3 0, E4 0} C_DIS
LIN {X 97.63, Y 31.573, Z 170.75, A 0, B 90, C 0, E1 0, E2 0, E3 0, E4 0} C_DIS
LIN {X 98.032, Y 28.529, Z 170.75, A 0, B 90, C 0, E1 0, E2 0, E3 0, E4 0} C_DIS
LIN {X 98.15, Y 25.461, Z 170.75, A 0, B 90, C 0, E1 0, E2 0, E3 0, E4 0} C_DIS
LIN {X 97.99, Y 22.395, Z 170.75, A 0, B 90, C 0, E1 0, E2 0, E3 0, E4 0} C_DIS
LIN {X 97.56, Y 19.355, Z 170.75, A 0, B 90, C 0, E1 0, E2 0, E3 0, E4 0} C_DIS
LIN {X 96.873, Y 16.362, Z 170.75, A 0, B 90, C 0, E1 0, E2 0, E3 0, E4 0} C_DIS
LIN {X 95.949, Y 13.434, Z 170.75, A 0, B 90, C 0, E1 0, E2 0, E3 0, E4 0} C_DIS
LIN {X 94.814, Y 10.58, Z 170.75, A 0, B 90, C 0, E1 0, E2 0, E3 0, E4 0} C_DIS
LIN {X 93.5, Y 7.805, Z 170.75, A 0, B 90, C 0, E1 0, E2 0, E3 0, E4 0} C_DIS
LIN {X 92.035, Y 5.106, Z 170.75, A 0, B 90, C 0, E1 0, E2 0, E3 0, E4 0} C_DIS
LIN {X 90.436, Y 2.485, Z 170.75, A 0, B 90, C 0, E1 0, E2 0, E3 0, E4 0} C_DIS
LIN {X 88.767, Y 0, Z 170.75, A 0, B 90, C 0, E1 0, E2 0, E3 0, E4 0} C_DIS
LIN {X 86.839, Y -2.046, Z 170.75, A 0, B 90, C 0, E1 0, E2 0, E3 0, E4 0} C_DIS
LIN {X 84.959, Y -4.474, Z 170.75, A 0, B 90, C 0, E1 0, E2 0, E3 0, E4 0} C_DIS
LIN {X 83.048, Y -6.878, Z 170.75, A 0, B 90, C 0, E1 0, E2 0, E3 0, E4 0} C_DIS
LIN {X 81.102, Y -9.254, Z 170.75, A 0, B 90, C 0, E1 0, E2 0, E3 0, E4 0} C_DIS
LIN {X 79.154, Y -11.629, Z 170.75, A 0, B 90, C 0, E1 0, E2 0, E3 0, E4 0} C_DIS
LIN {X 77.247, Y -14.037, Z 170.75, A 0, B 90, C 0, E1 0, E2 0, E3 0, E4 0} C_DIS
LIN {X 75.416, Y -16.502, Z 170.75, A 0, B 90, C 0, E1 0, E2 0, E3 0, E4 0} C_DIS
LIN {X 73.681, Y -19.036, Z 170.75, A 0, B 90, C 0, E1 0, E2 0, E3 0, E4 0} C_DIS
LIN {X 72.073, Y -21.652, Z 170.75, A 0, B 90, C 0, E1 0, E2 0, E3 0, E4 0} C_DIS
LIN {X 70.637, Y -24.367, Z 170.75, A 0, B 90, C 0, E1 0, E2 0, E3 0, E4 0} C_DIS
LIN {X 69.417, Y -27.184, Z 170.75, A 0, B 90, C 0, E1 0, E2 0, E3 0, E4 0} C_DIS
LIN {X 68.444, Y -30.097, Z 170.75, A 0, B 90, C 0, E1 0, E2 0, E3 0, E4 0} C_DIS
LIN {X 67.71, Y -33.078, Z 170.75, A 0, B 90, C 0, E1 0, E2 0, E3 0, E4 0} C_DIS
LIN {X 67.179, Y -36.103, Z 170.75, A 0, B 90, C 0, E1 0, E2 0, E3 0, E4 0} C_DIS
LIN {X 66.795, Y -39.15, Z 170.75, A 0, B 90, C 0, E1 0, E2 0, E3 0, E4 0} C_DIS
LIN {X 66.497, Y -42.207, Z 170.75, A 0, B 90, C 0, E1 0, E2 0, E3 0, E4 0} C_DIS
LIN {X 66.228, Y -45.266, Z 170.75, A 0, B 90, C 0, E1 0, E2 0, E3 0, E4 0} C_DIS
LIN {X 65.937, Y -48.324, Z 170.75, A 0, B 90, C 0, E1 0, E2 0, E3 0, E4 0} C_DIS
LIN {X 65.586, Y -51.375, Z 170.75, A 0, B 90, C 0, E1 0, E2 0, E3 0, E4 0} C_DIS
LIN {X 65.154, Y -54.416, Z 170.75, A 0, B 90, C 0, E1 0, E2 0, E3 0, E4 0} C_DIS
LIN {X 64.628, Y -57.442, Z 170.75, A 0, B 90, C 0, E1 0, E2 0, E3 0, E4 0} C_DIS
LIN {X 64.001, Y -60.448, Z 170.75, A 0, B 90, C 0, E1 0, E2 0, E3 0, E4 0} C_DIS
LIN {X 63.261, Y -63.429, Z 170.75, A 0, B 90, C 0, E1 0, E2 0, E3 0, E4 0} C_DIS
LIN {X 62.396, Y -66.375, Z 170.75, A 0, B 90, C 0, E1 0, E2 0, E3 0, E4 0} C_DIS
LIN {X 61.394, Y -69.278, Z 170.75, A 0, B 90, C 0, E1 0, E2 0, E3 0, E4 0} C_DIS
LIN {X 60.243, Y -72.126, Z 170.75, A 0, B 90, C 0, E1 0, E2 0, E3 0, E4 0} C_DIS
LIN {X 58.935, Y -74.904, Z 170.75, A 0, B 90, C 0, E1 0, E2 0, E3 0, E4 0} C_DIS
LIN {X 57.462, Y -77.598, Z 170.75, A 0, B 90, C 0, E1 0, E2 0, E3 0, E4 0} C_DIS
LIN {X 55.823, Y -80.195, Z 170.75, A 0, B 90, C 0, E1 0, E2 0, E3 0, E4 0} C_DIS
LIN {X 54.027, Y -82.686, Z 170.75, A 0, B 90, C 0, E1 0, E2 0, E3 0, E4 0} C_DIS
LIN {X 52.096, Y -85.074, Z 170.75, A 0, B 90, C 0, E1 0, E2 0, E3 0, E4 0} C_DIS
LIN {X 50.039, Y -87.354, Z 170.75, A 0, B 90, C 0, E1 0, E2 0, E3 0, E4 0} C_DIS
LIN {X 47.838, Y -89.496, Z 170.75, A 0, B 90, C 0, E1 0, E2 0, E3 0, E4 0} C_DIS
LIN {X 45.476, Y -91.458, Z 170.75, A 0, B 90, C 0, E1 0, E2 0, E3 0, E4 0} C_DIS
LIN {X 42.954, Y -93.209, Z 170.75, A 0, B 90, C 0, E1 0, E2 0, E3 0, E4 0} C_DIS
LIN {X 40.281, Y -94.72, Z 170.75, A 0, B 90, C 0, E1 0, E2 0, E3 0, E4 0} C_DIS
LIN {X 37.477, Y -95.969, Z 170.75, A 0, B 90, C 0, E1 0, E2 0, E3 0, E4 0} C_DIS
LIN {X 34.565, Y -96.942, Z 170.75, A 0, B 90, C 0, E1 0, E2 0, E3 0, E4 0} C_DIS
LIN {X 31.573, Y -97.63, Z 170.75, A 0, B 90, C 0, E1 0, E2 0, E3 0, E4 0} C_DIS
LIN {X 28.529, Y -98.032, Z 170.75, A 0, B 90, C 0, E1 0, E2 0, E3 0, E4 0} C_DIS
LIN {X 25.461, Y -98.15, Z 170.75, A 0, B 90, C 0, E1 0, E2 0, E3 0, E4 0} C_DIS
LIN {X 22.395, Y -97.99, Z 170.75, A 0, B 90, C 0, E1 0, E2 0, E3 0, E4 0} C_DIS
LIN {X 19.355, Y -97.56, Z 170.75, A 0, B 90, C 0, E1 0, E2 0, E3 0, E4 0} C_DIS
LIN {X 16.362, Y -96.873, Z 170.75, A 0, B 90, C 0, E1 0, E2 0, E3 0, E4 0} C_DIS
LIN {X 13.434, Y -95.949, Z 170.75, A 0, B 90, C 0, E1 0, E2 0, E3 0, E4 0} C_DIS
LIN {X 10.58, Y -94.814, Z 170.75, A 0, B 90, C 0, E1 0, E2 0, E3 0, E4 0} C_DIS
LIN {X 7.805, Y -93.5, Z 170.75, A 0, B 90, C 0, E1 0, E2 0, E3 0, E4 0} C_DIS
LIN {X 5.106, Y -92.035, Z 170.75, A 0, B 90, C 0, E1 0, E2 0, E3 0, E4 0} C_DIS
LIN {X 2.485, Y -90.436, Z 170.75, A 0, B 90, C 0, E1 0, E2 0, E3 0, E4 0} C_DIS
LIN {X 0, Y -88.767, Z 170.75, A 0, B 90, C 0, E1 0, E2 0, E3 0, E4 0} C_DIS
LIN {X -2.046, Y -86.839, Z 170.75, A 0, B 90, C 0, E1 0, E2 0, E3 0, E4 0} C_DIS
LIN {X -4.474, Y -84.959, Z 170.75, A 0, B 90, C 0, E1 0, E2 0, E3 0, E4 0} C_DIS
LIN {X -6.878, Y -83.048, Z 170.75, A 0, B 90, C 0, E1 0, E2 0, E3 0, E4 0} C_DIS
LIN {X -9.254, Y -81.102, Z 170.75, A 0, B 90, C 0, E1 0, E2 0, E3 0, E4 0} C_DIS
LIN {X -11.629, Y -79.154, Z 170.75, A 0, B 90, C 0, E1 0, E2 0, E3 0, E4 0} C_DIS
LIN {X -14.037, Y -77.247, Z 170.75, A 0, B 90, C 0, E1 0, E2 0, E3 0, E4 0} C_DIS
LIN {X -16.502, Y -75.416, Z 170.75, A 0, B 90, C 0, E1 0, E2 0, E3 0, E4 0} C_DIS
LIN {X -19.036, Y -73.681, Z 170.75, A 0, B 90, C 0, E1 0, E2 0, E3 0, E4 0} C_DIS
LIN {X -21.652, Y -72.073, Z 170.75, A 0, B 90, C 0, E1 0, E2 0, E3 0, E4 0} C_DIS
LIN {X -24.367, Y -70.637, Z 170.75, A 0, B 90, C 0, E1 0, E2 0, E3 0, E4 0} C_DIS
LIN {X -27.184, Y -69.417, Z 170.75, A 0, B 90, C 0, E1 0, E2 0, E3 0, E4 0} C_DIS
LIN {X -30.097, Y -68.444, Z 170.75, A 0, B 90, C 0, E1 0, E2 0, E3 0, E4 0} C_DIS
LIN {X -33.078, Y -67.71, Z 170.75, A 0, B 90, C 0, E1 0, E2 0, E3 0, E4 0} C_DIS
LIN {X -36.103, Y -67.179, Z 170.75, A 0, B 90, C 0, E1 0, E2 0, E3 0, E4 0} C_DIS
LIN {X -39.15, Y -66.795, Z 170.75, A 0, B 90, C 0, E1 0, E2 0, E3 0, E4 0} C_DIS
LIN {X -42.207, Y -66.497, Z 170.75, A 0, B 90, C 0, E1 0, E2 0, E3 0, E4 0} C_DIS
LIN {X -45.266, Y -66.228, Z 170.75, A 0, B 90, C 0, E1 0, E2 0, E3 0, E4 0} C_DIS
LIN {X -48.324, Y -65.937, Z 170.75, A 0, B 90, C 0, E1 0, E2 0, E3 0, E4 0} C_DIS
LIN {X -51.375, Y -65.586, Z 170.75, A 0, B 90, C 0, E1 0, E2 0, E3 0, E4 0} C_DIS
LIN {X -54.416, Y -65.154, Z 170.75, A 0, B 90, C 0, E1 0, E2 0, E3 0, E4 0} C_DIS
LIN {X -57.442, Y -64.628, Z 170.75, A 0, B 90, C 0, E1 0, E2 0, E3 0, E4 0} C_DIS
LIN {X -60.448, Y -64.001, Z 170.75, A 0, B 90, C 0, E1 0, E2 0, E3 0, E4 0} C_DIS
LIN {X -63.429, Y -63.261, Z 170.75, A 0, B 90, C 0, E1 0, E2 0, E3 0, E4 0} C_DIS
LIN {X -66.375, Y -62.396, Z 170.75, A 0, B 90, C 0, E1 0, E2 0, E3 0, E4 0} C_DIS
LIN {X -69.278, Y -61.394, Z 170.75, A 0, B 90, C 0, E1 0, E2 0, E3 0, E4 0} C_DIS
LIN {X -72.126, Y -60.243, Z 170.75, A 0, B 90, C 0, E1 0, E2 0, E3 0, E4 0} C_DIS
LIN {X -74.904, Y -58.935, Z 170.75, A 0, B 90, C 0, E1 0, E2 0, E3 0, E4 0} C_DIS
LIN {X -77.598, Y -57.462, Z 170.75, A 0, B 90, C 0, E1 0, E2 0, E3 0, E4 0} C_DIS
LIN {X -80.195, Y -55.823, Z 170.75, A 0, B 90, C 0, E1 0, E2 0, E3 0, E4 0} C_DIS
LIN {X -82.686, Y -54.027, Z 170.75, A 0, B 90, C 0, E1 0, E2 0, E3 0, E4 0} C_DIS
LIN {X -85.074, Y -52.096, Z 170.75, A 0, B 90, C 0, E1 0, E2 0, E3 0, E4 0} C_DIS
LIN {X -87.354, Y -50.039, Z 170.75, A 0, B 90, C 0, E1 0, E2 0, E3 0, E4 0} C_DIS
LIN {X -89.496, Y -47.838, Z 170.75, A 0, B 90, C 0, E1 0, E2 0, E3 0, E4 0} C_DIS
LIN {X -91.458, Y -45.476, Z 170.75, A 0, B 90, C 0, E1 0, E2 0, E3 0, E4 0} C_DIS
LIN {X -93.209, Y -42.954, Z 170.75, A 0, B 90, C 0, E1 0, E2 0, E3 0, E4 0} C_DIS
LIN {X -94.72, Y -40.281, Z 170.75, A 0, B 90, C 0, E1 0, E2 0, E3 0, E4 0} C_DIS
LIN {X -95.969, Y -37.477, Z 170.75, A 0, B 90, C 0, E1 0, E2 0, E3 0, E4 0} C_DIS
LIN {X -96.942, Y -34.565, Z 170.75, A 0, B 90, C 0, E1 0, E2 0, E3 0, E4 0} C_DIS
LIN {X -97.63, Y -31.573, Z 170.75, A 0, B 90, C 0, E1 0, E2 0, E3 0, E4 0} C_DIS
LIN {X -98.032, Y -28.529, Z 170.75, A 0, B 90, C 0, E1 0, E2 0, E3 0, E4 0} C_DIS
LIN {X -98.15, Y -25.461, Z 170.75, A 0, B 90, C 0, E1 0, E2 0, E3 0, E4 0} C_DIS
LIN {X -97.99, Y -22.395, Z 170.75, A 0, B 90, C 0, E1 0, E2 0, E3 0, E4 0} C_DIS
LIN {X -97.56, Y -19.355, Z 170.75, A 0, B 90, C 0, E1 0, E2 0, E3 0, E4 0} C_DIS
LIN {X -96.873, Y -16.362, Z 170.75, A 0, B 90, C 0, E1 0, E2 0, E3 0, E4 0} C_DIS
LIN {X -95.949, Y -13.434, Z 170.75, A 0, B 90, C 0, E1 0, E2 0, E3 0, E4 0} C_DIS
LIN {X -94.814, Y -10.58, Z 170.75, A 0, B 90, C 0, E1 0, E2 0, E3 0, E4 0} C_DIS
LIN {X -93.5, Y -7.805, Z 170.75, A 0, B 90, C 0, E1 0, E2 0, E3 0, E4 0} C_DIS
LIN {X -92.035, Y -5.106, Z 170.75, A 0, B 90, C 0, E1 0, E2 0, E3 0, E4 0} C_DIS
LIN {X -90.436, Y -2.485, Z 170.75, A 0, B 90, C 0, E1 0, E2 0, E3 0, E4 0} C_DIS
LIN {X -89.206, Y 0, Z 173.25, A 0, B 90, C 0, E1 0, E2 0, E3 0, E4 0} C_DIS
LIN {X -87.26, Y 2.045, Z 173.25, A 0, B 90, C 0, E1 0, E2 0, E3 0, E4 0} C_DIS
LIN {X -85.359, Y 4.472, Z 173.25, A 0, B 90, C 0, E1 0, E2 0, E3 0, E4 0} C_DIS
LIN {X -83.429, Y 6.878, Z 173.25, A 0, B 90, C 0, E1 0, E2 0, E3 0, E4 0} C_DIS
LIN {X -81.467, Y 9.258, Z 173.25, A 0, B 90, C 0, E1 0, E2 0, E3 0, E4 0} C_DIS
LIN {X -79.507, Y 11.64, Z 173.25, A 0, B 90, C 0, E1 0, E2 0, E3 0, E4 0} C_DIS
LIN {X -77.597, Y 14.061, Z 173.25, A 0, B 90, C 0, E1 0, E2 0, E3 0, E4 0} C_DIS
LIN {X -75.775, Y 16.549, Z 173.25, A 0, B 90, C 0, E1 0, E2 0, E3 0, E4 0} C_DIS
LIN {X -74.058, Y 19.111, Z 173.25, A 0, B 90, C 0, E1 0, E2 0, E3 0, E4 0} C_DIS
LIN {X -72.473, Y 21.756, Z 173.25, A 0, B 90, C 0, E1 0, E2 0, E3 0, E4 0} C_DIS
LIN {X -71.062, Y 24.499, Z 173.25, A 0, B 90, C 0, E1 0, E2 0, E3 0, E4 0} C_DIS
LIN {X -69.87, Y 27.342, Z 173.25, A 0, B 90, C 0, E1 0, E2 0, E3 0, E4 0} C_DIS
LIN {X -68.925, Y 30.277, Z 173.25, A 0, B 90, C 0, E1 0, E2 0, E3 0, E4 0} C_DIS
LIN {X -68.218, Y 33.279, Z 173.25, A 0, B 90, C 0, E1 0, E2 0, E3 0, E4 0} C_DIS
LIN {X -67.712, Y 36.321, Z 173.25, A 0, B 90, C 0, E1 0, E2 0, E3 0, E4 0} C_DIS
LIN {X -67.348, Y 39.384, Z 173.25, A 0, B 90, C 0, E1 0, E2 0, E3 0, E4 0} C_DIS
LIN {X -67.065, Y 42.455, Z 173.25, A 0, B 90, C 0, E1 0, E2 0, E3 0, E4 0} C_DIS
LIN {X -66.803, Y 45.528, Z 173.25, A 0, B 90, C 0, E1 0, E2 0, E3 0, E4 0} C_DIS
LIN {X -66.509, Y 48.598, Z 173.25, A 0, B 90, C 0, E1 0, E2 0, E3 0, E4 0} C_DIS
LIN {X -66.144, Y 51.661, Z 173.25, A 0, B 90, C 0, E1 0, E2 0, E3 0, E4 0} C_DIS
LIN {X -65.687, Y 54.711, Z 173.25, A 0, B 90, C 0, E1 0, E2 0, E3 0, E4 0} C_DIS
LIN {X -65.128, Y 57.744, Z 173.25, A 0, B 90, C 0, E1 0, E2 0, E3 0, E4 0} C_DIS
LIN {X -64.463, Y 60.756, Z 173.25, A 0, B 90, C 0, E1 0, E2 0, E3 0, E4 0} C_DIS
LIN {X -63.682, Y 63.739, Z 173.25, A 0, B 90, C 0, E1 0, E2 0, E3 0, E4 0} C_DIS
LIN {X -62.773, Y 66.686, Z 173.25, A 0, B 90, C 0, E1 0, E2 0, E3 0, E4 0} C_DIS
LIN {X -61.726, Y 69.587, Z 173.25, A 0, B 90, C 0, E1 0, E2 0, E3 0, E4 0} C_DIS
LIN {X -60.529, Y 72.429, Z 173.25, A 0, B 90, C 0, E1 0, E2 0, E3 0, E4 0} C_DIS
LIN {X -59.173, Y 75.199, Z 173.25, A 0, B 90, C 0, E1 0, E2 0, E3 0, E4 0} C_DIS
LIN {X -57.654, Y 77.883, Z 173.25, A 0, B 90, C 0, E1 0, E2 0, E3 0, E4 0} C_DIS
LIN {X -55.972, Y 80.468, Z 173.25, A 0, B 90, C 0, E1 0, E2 0, E3 0, E4 0} C_DIS
LIN {X -54.141, Y 82.949, Z 173.25, A 0, B 90, C 0, E1 0, E2 0, E3 0, E4 0} C_DIS
LIN {X -52.187, Y 85.335, Z 173.25, A 0, B 90, C 0, E1 0, E2 0, E3 0, E4 0} C_DIS
LIN {X -50.122, Y 87.626, Z 173.25, A 0, B 90, C 0, E1 0, E2 0, E3 0, E4 0} C_DIS
LIN {X -47.922, Y 89.786, Z 173.25, A 0, B 90, C 0, E1 0, E2 0, E3 0, E4 0} C_DIS
LIN {X -45.565, Y 91.774, Z 173.25, A 0, B 90, C 0, E1 0, E2 0, E3 0, E4 0} C_DIS
LIN {X -43.047, Y 93.554, Z 173.25, A 0, B 90, C 0, E1 0, E2 0, E3 0, E4 0} C_DIS
LIN {X -40.377, Y 95.097, Z 173.25, A 0, B 90, C 0, E1 0, E2 0, E3 0, E4 0} C_DIS
LIN {X -37.574, Y 96.379, Z 173.25, A 0, B 90, C 0, E1 0, E2 0, E3 0, E4 0} C_DIS
LIN {X -34.659, Y 97.384, Z 173.25, A 0, B 90, C 0, E1 0, E2 0, E3 0, E4 0} C_DIS
LIN {X -31.661, Y 98.104, Z 173.25, A 0, B 90, C 0, E1 0, E2 0, E3 0, E4 0} C_DIS
LIN {X -28.608, Y 98.534, Z 173.25, A 0, B 90, C 0, E1 0, E2 0, E3 0, E4 0} C_DIS
LIN {X -25.528, Y 98.676, Z 173.25, A 0, B 90, C 0, E1 0, E2 0, E3 0, E4 0} C_DIS
LIN {X -22.448, Y 98.533, Z 173.25, A 0, B 90, C 0, E1 0, E2 0, E3 0, E4 0} C_DIS
LIN {X -19.394, Y 98.112, Z 173.25, A 0, B 90, C 0, E1 0, E2 0, E3 0, E4 0} C_DIS
LIN {X -16.388, Y 97.424, Z 173.25, A 0, B 90, C 0, E1 0, E2 0, E3 0, E4 0} C_DIS
LIN {X -13.449, Y 96.491, Z 173.25, A 0, B 90, C 0, E1 0, E2 0, E3 0, E4 0} C_DIS
LIN {X -10.588, Y 95.34, Z 173.25, A 0, B 90, C 0, E1 0, E2 0, E3 0, E4 0} C_DIS
LIN {X -7.808, Y 94.006, Z 173.25, A 0, B 90, C 0, E1 0, E2 0, E3 0, E4 0} C_DIS
LIN {X -5.106, Y 92.519, Z 173.25, A 0, B 90, C 0, E1 0, E2 0, E3 0, E4 0} C_DIS
LIN {X -2.485, Y 90.896, Z 173.25, A 0, B 90, C 0, E1 0, E2 0, E3 0, E4 0} C_DIS
LIN {X 0, Y 89.206, Z 173.25, A 0, B 90, C 0, E1 0, E2 0, E3 0, E4 0} C_DIS
LIN {X 2.045, Y 87.26, Z 173.25, A 0, B 90, C 0, E1 0, E2 0, E3 0, E4 0} C_DIS
LIN {X 4.472, Y 85.359, Z 173.25, A 0, B 90, C 0, E1 0, E2 0, E3 0, E4 0} C_DIS
LIN {X 6.878, Y 83.429, Z 173.25, A 0, B 90, C 0, E1 0, E2 0, E3 0, E4 0} C_DIS
LIN {X 9.258, Y 81.467, Z 173.25, A 0, B 90, C 0, E1 0, E2 0, E3 0, E4 0} C_DIS
LIN {X 11.64, Y 79.507, Z 173.25, A 0, B 90, C 0, E1 0, E2 0, E3 0, E4 0} C_DIS
LIN {X 14.061, Y 77.597, Z 173.25, A 0, B 90, C 0, E1 0, E2 0, E3 0, E4 0} C_DIS
LIN {X 16.549, Y 75.775, Z 173.25, A 0, B 90, C 0, E1 0, E2 0, E3 0, E4 0} C_DIS
LIN {X 19.111, Y 74.058, Z 173.25, A 0, B 90, C 0, E1 0, E2 0, E3 0, E4 0} C_DIS
LIN {X 21.756, Y 72.473, Z 173.25, A 0, B 90, C 0, E1 0, E2 0, E3 0, E4 0} C_DIS
LIN {X 24.499, Y 71.062, Z 173.25, A 0, B 90, C 0, E1 0, E2 0, E3 0, E4 0} C_DIS
LIN {X 27.342, Y 69.87, Z 173.25, A 0, B 90, C 0, E1 0, E2 0, E3 0, E4 0} C_DIS
LIN {X 30.277, Y 68.925, Z 173.25, A 0, B 90, C 0, E1 0, E2 0, E3 0, E4 0} C_DIS
LIN {X 33.279, Y 68.218, Z 173.25, A 0, B 90, C 0, E1 0, E2 0, E3 0, E4 0} C_DIS
LIN {X 36.321, Y 67.712, Z 173.25, A 0, B 90, C 0, E1 0, E2 0, E3 0, E4 0} C_DIS
LIN {X 39.384, Y 67.348, Z 173.25, A 0, B 90, C 0, E1 0, E2 0, E3 0, E4 0} C_DIS
LIN {X 42.455, Y 67.065, Z 173.25, A 0, B 90, C 0, E1 0, E2 0, E3 0, E4 0} C_DIS
LIN {X 45.528, Y 66.803, Z 173.25, A 0, B 90, C 0, E1 0, E2 0, E3 0, E4 0} C_DIS
LIN {X 48.598, Y 66.509, Z 173.25, A 0, B 90, C 0, E1 0, E2 0, E3 0, E4 0} C_DIS
LIN {X 51.661, Y 66.144, Z 173.25, A 0, B 90, C 0, E1 0, E2 0, E3 0, E4 0} C_DIS
LIN {X 54.711, Y 65.687, Z 173.25, A 0, B 90, C 0, E1 0, E2 0, E3 0, E4 0} C_DIS
LIN {X 57.744, Y 65.128, Z 173.25, A 0, B 90, C 0, E1 0, E2 0, E3 0, E4 0} C_DIS
LIN {X 60.756, Y 64.463, Z 173.25, A 0, B 90, C 0, E1 0, E2 0, E3 0, E4 0} C_DIS
LIN {X 63.739, Y 63.682, Z 173.25, A 0, B 90, C 0, E1 0, E2 0, E3 0, E4 0} C_DIS
LIN {X 66.686, Y 62.773, Z 173.25, A 0, B 90, C 0, E1 0, E2 0, E3 0, E4 0} C_DIS
LIN {X 69.587, Y 61.726, Z 173.25, A 0, B 90, C 0, E1 0, E2 0, E3 0, E4 0} C_DIS
LIN {X 72.429, Y 60.529, Z 173.25, A 0, B 90, C 0, E1 0, E2 0, E3 0, E4 0} C_DIS
LIN {X 75.199, Y 59.173, Z 173.25, A 0, B 90, C 0, E1 0, E2 0, E3 0, E4 0} C_DIS
LIN {X 77.883, Y 57.654, Z 173.25, A 0, B 90, C 0, E1 0, E2 0, E3 0, E4 0} C_DIS
LIN {X 80.468, Y 55.972, Z 173.25, A 0, B 90, C 0, E1 0, E2 0, E3 0, E4 0} C_DIS
LIN {X 82.949, Y 54.141, Z 173.25, A 0, B 90, C 0, E1 0, E2 0, E3 0, E4 0} C_DIS
LIN {X 85.335, Y 52.187, Z 173.25, A 0, B 90, C 0, E1 0, E2 0, E3 0, E4 0} C_DIS
LIN {X 87.626, Y 50.122, Z 173.25, A 0, B 90, C 0, E1 0, E2 0, E3 0, E4 0} C_DIS
LIN {X 89.786, Y 47.922, Z 173.25, A 0, B 90, C 0, E1 0, E2 0, E3 0, E4 0} C_DIS
LIN {X 91.774, Y 45.565, Z 173.25, A 0, B 90, C 0, E1 0, E2 0, E3 0, E4 0} C_DIS
LIN {X 93.554, Y 43.047, Z 173.25, A 0, B 90, C 0, E1 0, E2 0, E3 0, E4 0} C_DIS
LIN {X 95.097, Y 40.377, Z 173.25, A 0, B 90, C 0, E1 0, E2 0, E3 0, E4 0} C_DIS
LIN {X 96.379, Y 37.574, Z 173.25, A 0, B 90, C 0, E1 0, E2 0, E3 0, E4 0} C_DIS
LIN {X 97.384, Y 34.659, Z 173.25, A 0, B 90, C 0, E1 0, E2 0, E3 0, E4 0} C_DIS
LIN {X 98.104, Y 31.661, Z 173.25, A 0, B 90, C 0, E1 0, E2 0, E3 0, E4 0} C_DIS
LIN {X 98.534, Y 28.608, Z 173.25, A 0, B 90, C 0, E1 0, E2 0, E3 0, E4 0} C_DIS
LIN {X 98.676, Y 25.528, Z 173.25, A 0, B 90, C 0, E1 0, E2 0, E3 0, E4 0} C_DIS
LIN {X 98.533, Y 22.448, Z 173.25, A 0, B 90, C 0, E1 0, E2 0, E3 0, E4 0} C_DIS
LIN {X 98.112, Y 19.394, Z 173.25, A 0, B 90, C 0, E1 0, E2 0, E3 0, E4 0} C_DIS
LIN {X 97.424, Y 16.388, Z 173.25, A 0, B 90, C 0, E1 0, E2 0, E3 0, E4 0} C_DIS
LIN {X 96.491, Y 13.449, Z 173.25, A 0, B 90, C 0, E1 0, E2 0, E3 0, E4 0} C_DIS
LIN {X 95.34, Y 10.588, Z 173.25, A 0, B 90, C 0, E1 0, E2 0, E3 0, E4 0} C_DIS
LIN {X 94.006, Y 7.808, Z 173.25, A 0, B 90, C 0, E1 0, E2 0, E3 0, E4 0} C_DIS
LIN {X 92.519, Y 5.106, Z 173.25, A 0, B 90, C 0, E1 0, E2 0, E3 0, E4 0} C_DIS
LIN {X 90.896, Y 2.485, Z 173.25, A 0, B 90, C 0, E1 0, E2 0, E3 0, E4 0} C_DIS
LIN {X 89.206, Y 0, Z 173.25, A 0, B 90, C 0, E1 0, E2 0, E3 0, E4 0} C_DIS
LIN {X 87.26, Y -2.045, Z 173.25, A 0, B 90, C 0, E1 0, E2 0, E3 0, E4 0} C_DIS
LIN {X 85.359, Y -4.472, Z 173.25, A 0, B 90, C 0, E1 0, E2 0, E3 0, E4 0} C_DIS
LIN {X 83.429, Y -6.878, Z 173.25, A 0, B 90, C 0, E1 0, E2 0, E3 0, E4 0} C_DIS
LIN {X 81.467, Y -9.258, Z 173.25, A 0, B 90, C 0, E1 0, E2 0, E3 0, E4 0} C_DIS
LIN {X 79.507, Y -11.64, Z 173.25, A 0, B 90, C 0, E1 0, E2 0, E3 0, E4 0} C_DIS
LIN {X 77.597, Y -14.061, Z 173.25, A 0, B 90, C 0, E1 0, E2 0, E3 0, E4 0} C_DIS
LIN {X 75.775, Y -16.549, Z 173.25, A 0, B 90, C 0, E1 0, E2 0, E3 0, E4 0} C_DIS
LIN {X 74.058, Y -19.111, Z 173.25, A 0, B 90, C 0, E1 0, E2 0, E3 0, E4 0} C_DIS
LIN {X 72.473, Y -21.756, Z 173.25, A 0, B 90, C 0, E1 0, E2 0, E3 0, E4 0} C_DIS
LIN {X 71.062, Y -24.499, Z 173.25, A 0, B 90, C 0, E1 0, E2 0, E3 0, E4 0} C_DIS
LIN {X 69.87, Y -27.342, Z 173.25, A 0, B 90, C 0, E1 0, E2 0, E3 0, E4 0} C_DIS
LIN {X 68.925, Y -30.277, Z 173.25, A 0, B 90, C 0, E1 0, E2 0, E3 0, E4 0} C_DIS
LIN {X 68.218, Y -33.279, Z 173.25, A 0, B 90, C 0, E1 0, E2 0, E3 0, E4 0} C_DIS
LIN {X 67.712, Y -36.321, Z 173.25, A 0, B 90, C 0, E1 0, E2 0, E3 0, E4 0} C_DIS
LIN {X 67.348, Y -39.384, Z 173.25, A 0, B 90, C 0, E1 0, E2 0, E3 0, E4 0} C_DIS
LIN {X 67.065, Y -42.455, Z 173.25, A 0, B 90, C 0, E1 0, E2 0, E3 0, E4 0} C_DIS
LIN {X 66.803, Y -45.528, Z 173.25, A 0, B 90, C 0, E1 0, E2 0, E3 0, E4 0} C_DIS
LIN {X 66.509, Y -48.598, Z 173.25, A 0, B 90, C 0, E1 0, E2 0, E3 0, E4 0} C_DIS
LIN {X 66.144, Y -51.661, Z 173.25, A 0, B 90, C 0, E1 0, E2 0, E3 0, E4 0} C_DIS
LIN {X 65.687, Y -54.711, Z 173.25, A 0, B 90, C 0, E1 0, E2 0, E3 0, E4 0} C_DIS
LIN {X 65.128, Y -57.744, Z 173.25, A 0, B 90, C 0, E1 0, E2 0, E3 0, E4 0} C_DIS
LIN {X 64.463, Y -60.756, Z 173.25, A 0, B 90, C 0, E1 0, E2 0, E3 0, E4 0} C_DIS
LIN {X 63.682, Y -63.739, Z 173.25, A 0, B 90, C 0, E1 0, E2 0, E3 0, E4 0} C_DIS
LIN {X 62.773, Y -66.686, Z 173.25, A 0, B 90, C 0, E1 0, E2 0, E3 0, E4 0} C_DIS
LIN {X 61.726, Y -69.587, Z 173.25, A 0, B 90, C 0, E1 0, E2 0, E3 0, E4 0} C_DIS
LIN {X 60.529, Y -72.429, Z 173.25, A 0, B 90, C 0, E1 0, E2 0, E3 0, E4 0} C_DIS
LIN {X 59.173, Y -75.199, Z 173.25, A 0, B 90, C 0, E1 0, E2 0, E3 0, E4 0} C_DIS
LIN {X 57.654, Y -77.883, Z 173.25, A 0, B 90, C 0, E1 0, E2 0, E3 0, E4 0} C_DIS
LIN {X 55.972, Y -80.468, Z 173.25, A 0, B 90, C 0, E1 0, E2 0, E3 0, E4 0} C_DIS
LIN {X 54.141, Y -82.949, Z 173.25, A 0, B 90, C 0, E1 0, E2 0, E3 0, E4 0} C_DIS
LIN {X 52.187, Y -85.335, Z 173.25, A 0, B 90, C 0, E1 0, E2 0, E3 0, E4 0} C_DIS
LIN {X 50.122, Y -87.626, Z 173.25, A 0, B 90, C 0, E1 0, E2 0, E3 0, E4 0} C_DIS
LIN {X 47.922, Y -89.786, Z 173.25, A 0, B 90, C 0, E1 0, E2 0, E3 0, E4 0} C_DIS
LIN {X 45.565, Y -91.774, Z 173.25, A 0, B 90, C 0, E1 0, E2 0, E3 0, E4 0} C_DIS
LIN {X 43.047, Y -93.554, Z 173.25, A 0, B 90, C 0, E1 0, E2 0, E3 0, E4 0} C_DIS
LIN {X 40.377, Y -95.097, Z 173.25, A 0, B 90, C 0, E1 0, E2 0, E3 0, E4 0} C_DIS
LIN {X 37.574, Y -96.379, Z 173.25, A 0, B 90, C 0, E1 0, E2 0, E3 0, E4 0} C_DIS
LIN {X 34.659, Y -97.384, Z 173.25, A 0, B 90, C 0, E1 0, E2 0, E3 0, E4 0} C_DIS
LIN {X 31.661, Y -98.104, Z 173.25, A 0, B 90, C 0, E1 0, E2 0, E3 0, E4 0} C_DIS
LIN {X 28.608, Y -98.534, Z 173.25, A 0, B 90, C 0, E1 0, E2 0, E3 0, E4 0} C_DIS
LIN {X 25.528, Y -98.676, Z 173.25, A 0, B 90, C 0, E1 0, E2 0, E3 0, E4 0} C_DIS
LIN {X 22.448, Y -98.533, Z 173.25, A 0, B 90, C 0, E1 0, E2 0, E3 0, E4 0} C_DIS
LIN {X 19.394, Y -98.112, Z 173.25, A 0, B 90, C 0, E1 0, E2 0, E3 0, E4 0} C_DIS
LIN {X 16.388, Y -97.424, Z 173.25, A 0, B 90, C 0, E1 0, E2 0, E3 0, E4 0} C_DIS
LIN {X 13.449, Y -96.491, Z 173.25, A 0, B 90, C 0, E1 0, E2 0, E3 0, E4 0} C_DIS
LIN {X 10.588, Y -95.34, Z 173.25, A 0, B 90, C 0, E1 0, E2 0, E3 0, E4 0} C_DIS
LIN {X 7.808, Y -94.006, Z 173.25, A 0, B 90, C 0, E1 0, E2 0, E3 0, E4 0} C_DIS
LIN {X 5.106, Y -92.519, Z 173.25, A 0, B 90, C 0, E1 0, E2 0, E3 0, E4 0} C_DIS
LIN {X 2.485, Y -90.896, Z 173.25, A 0, B 90, C 0, E1 0, E2 0, E3 0, E4 0} C_DIS
LIN {X 0, Y -89.206, Z 173.25, A 0, B 90, C 0, E1 0, E2 0, E3 0, E4 0} C_DIS
LIN {X -2.045, Y -87.26, Z 173.25, A 0, B 90, C 0, E1 0, E2 0, E3 0, E4 0} C_DIS
LIN {X -4.472, Y -85.359, Z 173.25, A 0, B 90, C 0, E1 0, E2 0, E3 0, E4 0} C_DIS
LIN {X -6.878, Y -83.429, Z 173.25, A 0, B 90, C 0, E1 0, E2 0, E3 0, E4 0} C_DIS
LIN {X -9.258, Y -81.467, Z 173.25, A 0, B 90, C 0, E1 0, E2 0, E3 0, E4 0} C_DIS
LIN {X -11.64, Y -79.507, Z 173.25, A 0, B 90, C 0, E1 0, E2 0, E3 0, E4 0} C_DIS
LIN {X -14.061, Y -77.597, Z 173.25, A 0, B 90, C 0, E1 0, E2 0, E3 0, E4 0} C_DIS
LIN {X -16.549, Y -75.775, Z 173.25, A 0, B 90, C 0, E1 0, E2 0, E3 0, E4 0} C_DIS
LIN {X -19.111, Y -74.058, Z 173.25, A 0, B 90, C 0, E1 0, E2 0, E3 0, E4 0} C_DIS
LIN {X -21.756, Y -72.473, Z 173.25, A 0, B 90, C 0, E1 0, E2 0, E3 0, E4 0} C_DIS
LIN {X -24.499, Y -71.062, Z 173.25, A 0, B 90, C 0, E1 0, E2 0, E3 0, E4 0} C_DIS
LIN {X -27.342, Y -69.87, Z 173.25, A 0, B 90, C 0, E1 0, E2 0, E3 0, E4 0} C_DIS
LIN {X -30.277, Y -68.925, Z 173.25, A 0, B 90, C 0, E1 0, E2 0, E3 0, E4 0} C_DIS
LIN {X -33.279, Y -68.218, Z 173.25, A 0, B 90, C 0, E1 0, E2 0, E3 0, E4 0} C_DIS
LIN {X -36.321, Y -67.712, Z 173.25, A 0, B 90, C 0, E1 0, E2 0, E3 0, E4 0} C_DIS
LIN {X -39.384, Y -67.348, Z 173.25, A 0, B 90, C 0, E1 0, E2 0, E3 0, E4 0} C_DIS
LIN {X -42.455, Y -67.065, Z 173.25, A 0, B 90, C 0, E1 0, E2 0, E3 0, E4 0} C_DIS
LIN {X -45.528, Y -66.803, Z 173.25, A 0, B 90, C 0, E1 0, E2 0, E3 0, E4 0} C_DIS
LIN {X -48.598, Y -66.509, Z 173.25, A 0, B 90, C 0, E1 0, E2 0, E3 0, E4 0} C_DIS
LIN {X -51.661, Y -66.144, Z 173.25, A 0, B 90, C 0, E1 0, E2 0, E3 0, E4 0} C_DIS
LIN {X -54.711, Y -65.687, Z 173.25, A 0, B 90, C 0, E1 0, E2 0, E3 0, E4 0} C_DIS
LIN {X -57.744, Y -65.128, Z 173.25, A 0, B 90, C 0, E1 0, E2 0, E3 0, E4 0} C_DIS
LIN {X -60.756, Y -64.463, Z 173.25, A 0, B 90, C 0, E1 0, E2 0, E3 0, E4 0} C_DIS
LIN {X -63.739, Y -63.682, Z 173.25, A 0, B 90, C 0, E1 0, E2 0, E3 0, E4 0} C_DIS
LIN {X -66.686, Y -62.773, Z 173.25, A 0, B 90, C 0, E1 0, E2 0, E3 0, E4 0} C_DIS
LIN {X -69.587, Y -61.726, Z 173.25, A 0, B 90, C 0, E1 0, E2 0, E3 0, E4 0} C_DIS
LIN {X -72.429, Y -60.529, Z 173.25, A 0, B 90, C 0, E1 0, E2 0, E3 0, E4 0} C_DIS
LIN {X -75.199, Y -59.173, Z 173.25, A 0, B 90, C 0, E1 0, E2 0, E3 0, E4 0} C_DIS
LIN {X -77.883, Y -57.654, Z 173.25, A 0, B 90, C 0, E1 0, E2 0, E3 0, E4 0} C_DIS
LIN {X -80.468, Y -55.972, Z 173.25, A 0, B 90, C 0, E1 0, E2 0, E3 0, E4 0} C_DIS
LIN {X -82.949, Y -54.141, Z 173.25, A 0, B 90, C 0, E1 0, E2 0, E3 0, E4 0} C_DIS
LIN {X -85.335, Y -52.187, Z 173.25, A 0, B 90, C 0, E1 0, E2 0, E3 0, E4 0} C_DIS
LIN {X -87.626, Y -50.122, Z 173.25, A 0, B 90, C 0, E1 0, E2 0, E3 0, E4 0} C_DIS
LIN {X -89.786, Y -47.922, Z 173.25, A 0, B 90, C 0, E1 0, E2 0, E3 0, E4 0} C_DIS
LIN {X -91.774, Y -45.565, Z 173.25, A 0, B 90, C 0, E1 0, E2 0, E3 0, E4 0} C_DIS
LIN {X -93.554, Y -43.047, Z 173.25, A 0, B 90, C 0, E1 0, E2 0, E3 0, E4 0} C_DIS
LIN {X -95.097, Y -40.377, Z 173.25, A 0, B 90, C 0, E1 0, E2 0, E3 0, E4 0} C_DIS
LIN {X -96.379, Y -37.574, Z 173.25, A 0, B 90, C 0, E1 0, E2 0, E3 0, E4 0} C_DIS
LIN {X -97.384, Y -34.659, Z 173.25, A 0, B 90, C 0, E1 0, E2 0, E3 0, E4 0} C_DIS
LIN {X -98.104, Y -31.661, Z 173.25, A 0, B 90, C 0, E1 0, E2 0, E3 0, E4 0} C_DIS
LIN {X -98.534, Y -28.608, Z 173.25, A 0, B 90, C 0, E1 0, E2 0, E3 0, E4 0} C_DIS
LIN {X -98.676, Y -25.528, Z 173.25, A 0, B 90, C 0, E1 0, E2 0, E3 0, E4 0} C_DIS
LIN {X -98.533, Y -22.448, Z 173.25, A 0, B 90, C 0, E1 0, E2 0, E3 0, E4 0} C_DIS
LIN {X -98.112, Y -19.394, Z 173.25, A 0, B 90, C 0, E1 0, E2 0, E3 0, E4 0} C_DIS
LIN {X -97.424, Y -16.388, Z 173.25, A 0, B 90, C 0, E1 0, E2 0, E3 0, E4 0} C_DIS
LIN {X -96.491, Y -13.449, Z 173.25, A 0, B 90, C 0, E1 0, E2 0, E3 0, E4 0} C_DIS
LIN {X -95.34, Y -10.588, Z 173.25, A 0, B 90, C 0, E1 0, E2 0, E3 0, E4 0} C_DIS
LIN {X -94.006, Y -7.808, Z 173.25, A 0, B 90, C 0, E1 0, E2 0, E3 0, E4 0} C_DIS
LIN {X -92.519, Y -5.106, Z 173.25, A 0, B 90, C 0, E1 0, E2 0, E3 0, E4 0} C_DIS
LIN {X -90.896, Y -2.485, Z 173.25, A 0, B 90, C 0, E1 0, E2 0, E3 0, E4 0} C_DIS
LIN {X -89.655, Y 0, Z 175.75, A 0, B 90, C 0, E1 0, E2 0, E3 0, E4 0} C_DIS
LIN {X -87.691, Y 2.044, Z 175.75, A 0, B 90, C 0, E1 0, E2 0, E3 0, E4 0} C_DIS
LIN {X -85.769, Y 4.472, Z 175.75, A 0, B 90, C 0, E1 0, E2 0, E3 0, E4 0} C_DIS
LIN {X -83.82, Y 6.88, Z 175.75, A 0, B 90, C 0, E1 0, E2 0, E3 0, E4 0} C_DIS
LIN {X -81.841, Y 9.263, Z 175.75, A 0, B 90, C 0, E1 0, E2 0, E3 0, E4 0} C_DIS
LIN {X -79.87, Y 11.652, Z 175.75, A 0, B 90, C 0, E1 0, E2 0, E3 0, E4 0} C_DIS
LIN {X -77.957, Y 14.088, Z 175.75, A 0, B 90, C 0, E1 0, E2 0, E3 0, E4 0} C_DIS
LIN {X -76.144, Y 16.6, Z 175.75, A 0, B 90, C 0, E1 0, E2 0, E3 0, E4 0} C_DIS
LIN {X -74.446, Y 19.19, Z 175.75, A 0, B 90, C 0, E1 0, E2 0, E3 0, E4 0} C_DIS
LIN {X -72.885, Y 21.865, Z 175.75, A 0, B 90, C 0, E1 0, E2 0, E3 0, E4 0} C_DIS
LIN {X -71.502, Y 24.636, Z 175.75, A 0, B 90, C 0, E1 0, E2 0, E3 0, E4 0} C_DIS
LIN {X -70.34, Y 27.506, Z 175.75, A 0, B 90, C 0, E1 0, E2 0, E3 0, E4 0} C_DIS
LIN {X -69.424, Y 30.464, Z 175.75, A 0, B 90, C 0, E1 0, E2 0, E3 0, E4 0} C_DIS
LIN {X -68.745, Y 33.486, Z 175.75, A 0, B 90, C 0, E1 0, E2 0, E3 0, E4 0} C_DIS
LIN {X -68.265, Y 36.546, Z 175.75, A 0, B 90, C 0, E1 0, E2 0, E3 0, E4 0} C_DIS
LIN {X -67.921, Y 39.624, Z 175.75, A 0, B 90, C 0, E1 0, E2 0, E3 0, E4 0} C_DIS
LIN {X -67.653, Y 42.71, Z 175.75, A 0, B 90, C 0, E1 0, E2 0, E3 0, E4 0} C_DIS
LIN {X -67.397, Y 45.797, Z 175.75, A 0, B 90, C 0, E1 0, E2 0, E3 0, E4 0} C_DIS
LIN {X -67.1, Y 48.88, Z 175.75, A 0, B 90, C 0, E1 0, E2 0, E3 0, E4 0} C_DIS
LIN {X -66.72, Y 51.954, Z 175.75, A 0, B 90, C 0, E1 0, E2 0, E3 0, E4 0} C_DIS
LIN {X -66.237, Y 55.014, Z 175.75, A 0, B 90, C 0, E1 0, E2 0, E3 0, E4 0} C_DIS
LIN {X -65.645, Y 58.054, Z 175.75, A 0, B 90, C 0, E1 0, E2 0, E3 0, E4 0} C_DIS
LIN {X -64.94, Y 61.07, Z 175.75, A 0, B 90, C 0, E1 0, E2 0, E3 0, E4 0} C_DIS
LIN {X -64.115, Y 64.056, Z 175.75, A 0, B 90, C 0, E1 0, E2 0, E3 0, E4 0} C_DIS
LIN {X -63.16, Y 67.002, Z 175.75, A 0, B 90, C 0, E1 0, E2 0, E3 0, E4 0} C_DIS
LIN {X -62.065, Y 69.899, Z 175.75, A 0, B 90, C 0, E1 0, E2 0, E3 0, E4 0} C_DIS
LIN {X -60.819, Y 72.735, Z 175.75, A 0, B 90, C 0, E1 0, E2 0, E3 0, E4 0} C_DIS
LIN {X -59.415, Y 75.495, Z 175.75, A 0, B 90, C 0, E1 0, E2 0, E3 0, E4 0} C_DIS
LIN {X -57.848, Y 78.167, Z 175.75, A 0, B 90, C 0, E1 0, E2 0, E3 0, E4 0} C_DIS
LIN {X -56.122, Y 80.739, Z 175.75, A 0, B 90, C 0, E1 0, E2 0, E3 0, E4 0} C_DIS
LIN {X -54.255, Y 83.21, Z 175.75, A 0, B 90, C 0, E1 0, E2 0, E3 0, E4 0} C_DIS
LIN {X -52.278, Y 85.594, Z 175.75, A 0, B 90, C 0, E1 0, E2 0, E3 0, E4 0} C_DIS
LIN {X -50.205, Y 87.896, Z 175.75, A 0, B 90, C 0, E1 0, E2 0, E3 0, E4 0} C_DIS
LIN {X -48.006, Y 90.076, Z 175.75, A 0, B 90, C 0, E1 0, E2 0, E3 0, E4 0} C_DIS
LIN {X -45.653, Y 92.09, Z 175.75, A 0, B 90, C 0, E1 0, E2 0, E3 0, E4 0} C_DIS
LIN {X -43.141, Y 93.9, Z 175.75, A 0, B 90, C 0, E1 0, E2 0, E3 0, E4 0} C_DIS
LIN {X -40.475, Y 95.475, Z 175.75, A 0, B 90, C 0, E1 0, E2 0, E3 0, E4 0} C_DIS
LIN {X -37.672, Y 96.792, Z 175.75, A 0, B 90, C 0, E1 0, E2 0, E3 0, E4 0} C_DIS
LIN {X -34.756, Y 97.831, Z 175.75, A 0, B 90, C 0, E1 0, E2 0, E3 0, E4 0} C_DIS
LIN {X -31.752, Y 98.583, Z 175.75, A 0, B 90, C 0, E1 0, E2 0, E3 0, E4 0} C_DIS
LIN {X -28.69, Y 99.042, Z 175.75, A 0, B 90, C 0, E1 0, E2 0, E3 0, E4 0} C_DIS
LIN {X -25.598, Y 99.209, Z 175.75, A 0, B 90, C 0, E1 0, E2 0, E3 0, E4 0} C_DIS
LIN {X -22.504, Y 99.085, Z 175.75, A 0, B 90, C 0, E1 0, E2 0, E3 0, E4 0} C_DIS
LIN {X -19.435, Y 98.674, Z 175.75, A 0, B 90, C 0, E1 0, E2 0, E3 0, E4 0} C_DIS
LIN {X -16.416, Y 97.985, Z 175.75, A 0, B 90, C 0, E1 0, E2 0, E3 0, E4 0} C_DIS
LIN {X -13.466, Y 97.042, Z 175.75, A 0, B 90, C 0, E1 0, E2 0, E3 0, E4 0} C_DIS
LIN {X -10.597, Y 95.876, Z 175.75, A 0, B 90, C 0, E1 0, E2 0, E3 0, E4 0} C_DIS
LIN {X -7.812, Y 94.522, Z 175.75, A 0, B 90, C 0, E1 0, E2 0, E3 0, E4 0} C_DIS
LIN {X -5.107, Y 93.013, Z 175.75, A 0, B 90, C 0, E1 0, E2 0, E3 0, E4 0} C_DIS
LIN {X -2.485, Y 91.367, Z 175.75, A 0, B 90, C 0, E1 0, E2 0, E3 0, E4 0} C_DIS
LIN {X 0, Y 89.655, Z 175.75, A 0, B 90, C 0, E1 0, E2 0, E3 0, E4 0} C_DIS
LIN {X 2.044, Y 87.691, Z 175.75, A 0, B 90, C 0, E1 0, E2 0, E3 0, E4 0} C_DIS
LIN {X 4.472, Y 85.769, Z 175.75, A 0, B 90, C 0, E1 0, E2 0, E3 0, E4 0} C_DIS
LIN {X 6.88, Y 83.82, Z 175.75, A 0, B 90, C 0, E1 0, E2 0, E3 0, E4 0} C_DIS
LIN {X 9.263, Y 81.841, Z 175.75, A 0, B 90, C 0, E1 0, E2 0, E3 0, E4 0} C_DIS
LIN {X 11.652, Y 79.87, Z 175.75, A 0, B 90, C 0, E1 0, E2 0, E3 0, E4 0} C_DIS
LIN {X 14.088, Y 77.957, Z 175.75, A 0, B 90, C 0, E1 0, E2 0, E3 0, E4 0} C_DIS
LIN {X 16.6, Y 76.144, Z 175.75, A 0, B 90, C 0, E1 0, E2 0, E3 0, E4 0} C_DIS
LIN {X 19.19, Y 74.446, Z 175.75, A 0, B 90, C 0, E1 0, E2 0, E3 0, E4 0} C_DIS
LIN {X 21.865, Y 72.885, Z 175.75, A 0, B 90, C 0, E1 0, E2 0, E3 0, E4 0} C_DIS
LIN {X 24.636, Y 71.502, Z 175.75, A 0, B 90, C 0, E1 0, E2 0, E3 0, E4 0} C_DIS
LIN {X 27.506, Y 70.34, Z 175.75, A 0, B 90, C 0, E1 0, E2 0, E3 0, E4 0} C_DIS
LIN {X 30.464, Y 69.424, Z 175.75, A 0, B 90, C 0, E1 0, E2 0, E3 0, E4 0} C_DIS
LIN {X 33.486, Y 68.745, Z 175.75, A 0, B 90, C 0, E1 0, E2 0, E3 0, E4 0} C_DIS
LIN {X 36.546, Y 68.265, Z 175.75, A 0, B 90, C 0, E1 0, E2 0, E3 0, E4 0} C_DIS
LIN {X 39.624, Y 67.921, Z 175.75, A 0, B 90, C 0, E1 0, E2 0, E3 0, E4 0} C_DIS
LIN {X 42.71, Y 67.653, Z 175.75, A 0, B 90, C 0, E1 0, E2 0, E3 0, E4 0} C_DIS
LIN {X 45.797, Y 67.397, Z 175.75, A 0, B 90, C 0, E1 0, E2 0, E3 0, E4 0} C_DIS
LIN {X 48.88, Y 67.1, Z 175.75, A 0, B 90, C 0, E1 0, E2 0, E3 0, E4 0} C_DIS
LIN {X 51.954, Y 66.72, Z 175.75, A 0, B 90, C 0, E1 0, E2 0, E3 0, E4 0} C_DIS
LIN {X 55.014, Y 66.237, Z 175.75, A 0, B 90, C 0, E1 0, E2 0, E3 0, E4 0} C_DIS
LIN {X 58.054, Y 65.645, Z 175.75, A 0, B 90, C 0, E1 0, E2 0, E3 0, E4 0} C_DIS
LIN {X 61.07, Y 64.94, Z 175.75, A 0, B 90, C 0, E1 0, E2 0, E3 0, E4 0} C_DIS
LIN {X 64.056, Y 64.115, Z 175.75, A 0, B 90, C 0, E1 0, E2 0, E3 0, E4 0} C_DIS
LIN {X 67.002, Y 63.16, Z 175.75, A 0, B 90, C 0, E1 0, E2 0, E3 0, E4 0} C_DIS
LIN {X 69.899, Y 62.065, Z 175.75, A 0, B 90, C 0, E1 0, E2 0, E3 0, E4 0} C_DIS
LIN {X 72.735, Y 60.819, Z 175.75, A 0, B 90, C 0, E1 0, E2 0, E3 0, E4 0} C_DIS
LIN {X 75.495, Y 59.415, Z 175.75, A 0, B 90, C 0, E1 0, E2 0, E3 0, E4 0} C_DIS
LIN {X 78.167, Y 57.848, Z 175.75, A 0, B 90, C 0, E1 0, E2 0, E3 0, E4 0} C_DIS
LIN {X 80.739, Y 56.122, Z 175.75, A 0, B 90, C 0, E1 0, E2 0, E3 0, E4 0} C_DIS
LIN {X 83.21, Y 54.255, Z 175.75, A 0, B 90, C 0, E1 0, E2 0, E3 0, E4 0} C_DIS
LIN {X 85.594, Y 52.278, Z 175.75, A 0, B 90, C 0, E1 0, E2 0, E3 0, E4 0} C_DIS
LIN {X 87.896, Y 50.205, Z 175.75, A 0, B 90, C 0, E1 0, E2 0, E3 0, E4 0} C_DIS
LIN {X 90.076, Y 48.006, Z 175.75, A 0, B 90, C 0, E1 0, E2 0, E3 0, E4 0} C_DIS
LIN {X 92.09, Y 45.653, Z 175.75, A 0, B 90, C 0, E1 0, E2 0, E3 0, E4 0} C_DIS
LIN {X 93.9, Y 43.141, Z 175.75, A 0, B 90, C 0, E1 0, E2 0, E3 0, E4 0} C_DIS
LIN {X 95.475, Y 40.475, Z 175.75, A 0, B 90, C 0, E1 0, E2 0, E3 0, E4 0} C_DIS
